// TIA Portal V17 export
// export: Created 2023-09-11T12:03:28.587249Z, ExportSetting WithDefaults, DisplayName Totally Integrated Automation Portal, DisplayVersion V17 Update 6, DisplayName TIA Portal Openness, DisplayVersion V17 Update 6, DisplayName TIA Portal Teamcenter Gateway, DisplayVersion V17 Update 6, DisplayName TIA Portal Version Control Interface, DisplayVersion V17, DisplayName Simotion SCOUT TIA, DisplayVersion 5.4.3.0, DisplayName TIA Portal Test Suite Advanced, DisplayVersion V17 Update 1, DisplayName SIMOCODE ES, DisplayVersion V17 Update 5, DisplayName SINAMICS Startdrive Advanced, DisplayVersion V17 SP1, DisplayName SINAMICS Startdrive G130, G150, S120, S150, SINAMICS MV, S210, DisplayVersion V17 SP1, DisplayName SINAMICS Startdrive G110M, G120, G120C, G120D, G120P, G115D, DisplayVersion V17 SP1, DisplayName SIRIUS Safety ES, DisplayVersion V17 Update 5, DisplayName STEP 7 Professional, DisplayVersion V17 Update 6, DisplayName STEP 7 CFC, DisplayVersion V17 Update 1, DisplayName STEP 7 Safety, DisplayVersion V17 Update 6, DisplayName WinCC Advanced, DisplayVersion V17 Update 6, DisplayName SIMATIC Visualization Architect, DisplayVersion V17 Update 5
FUNCTION "03_Zone Cumulative" : Void   // FC4, F_FBD
{ S7_Optimized_Access := 'TRUE' }
VERSION : 0.1
// stored: AutoNumber true, IsIECCheckEnabled false, UDAEnableTagReadback false
BEGIN

REGION Network 1: S1 PB - ^S1 | Sorter COY Upper [=SC01]
   // 251 - 500 Inputs
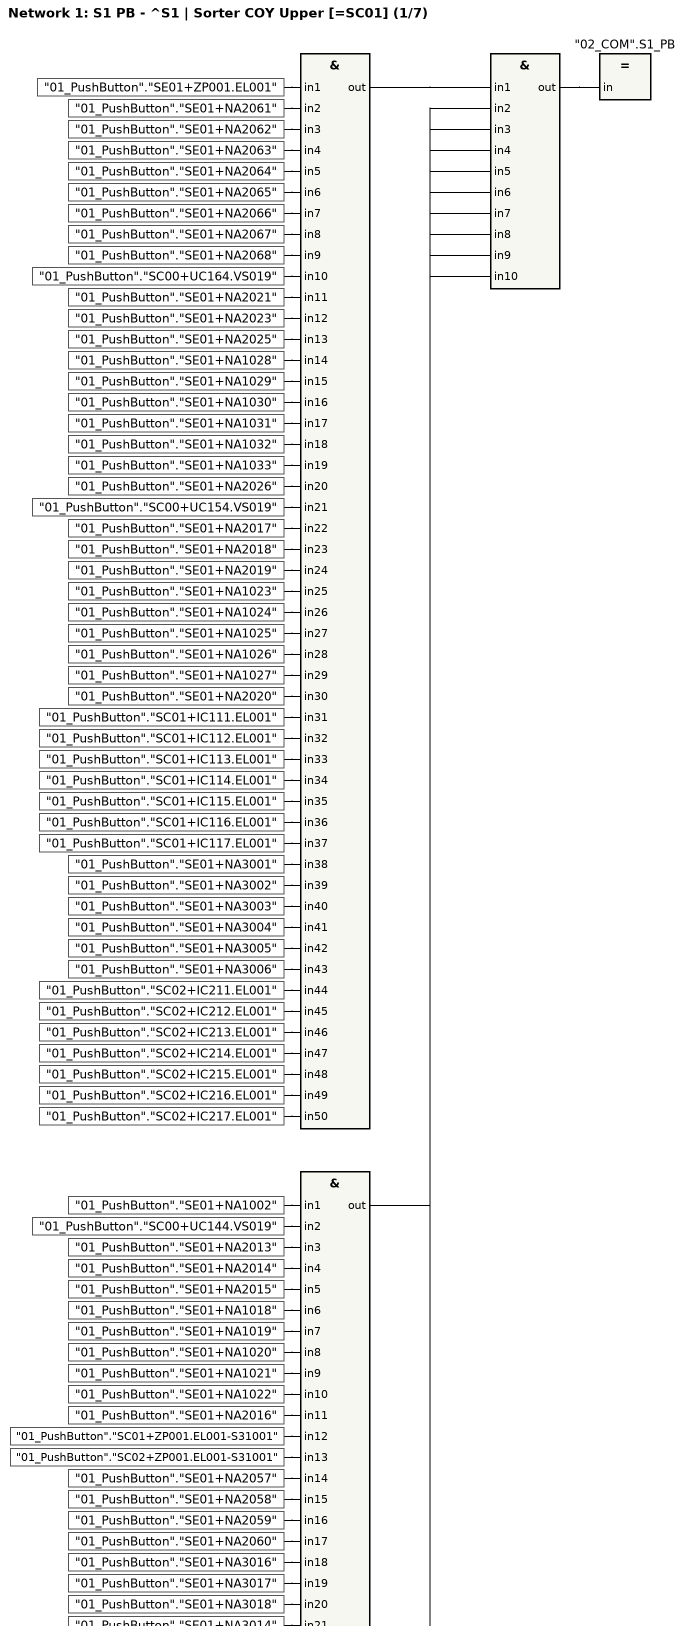
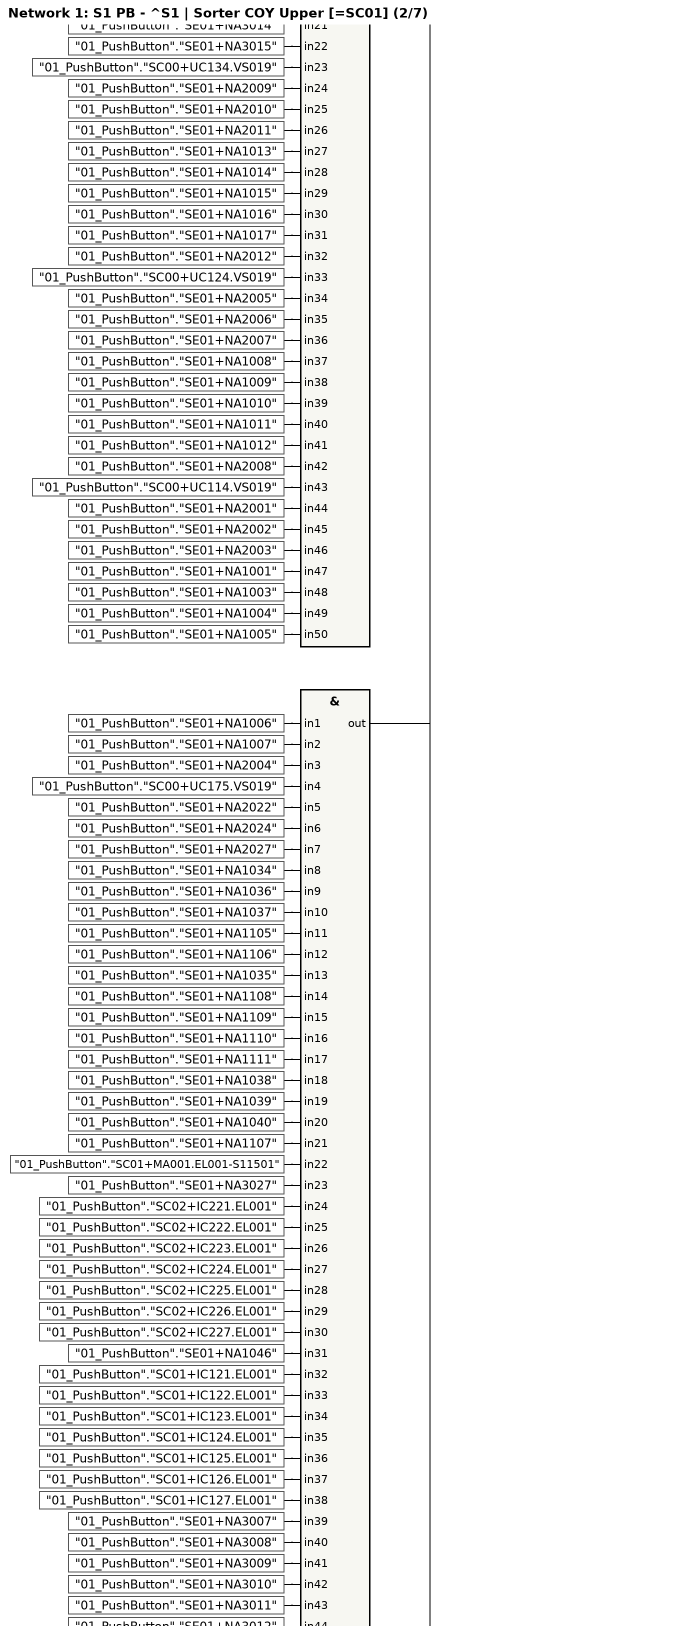
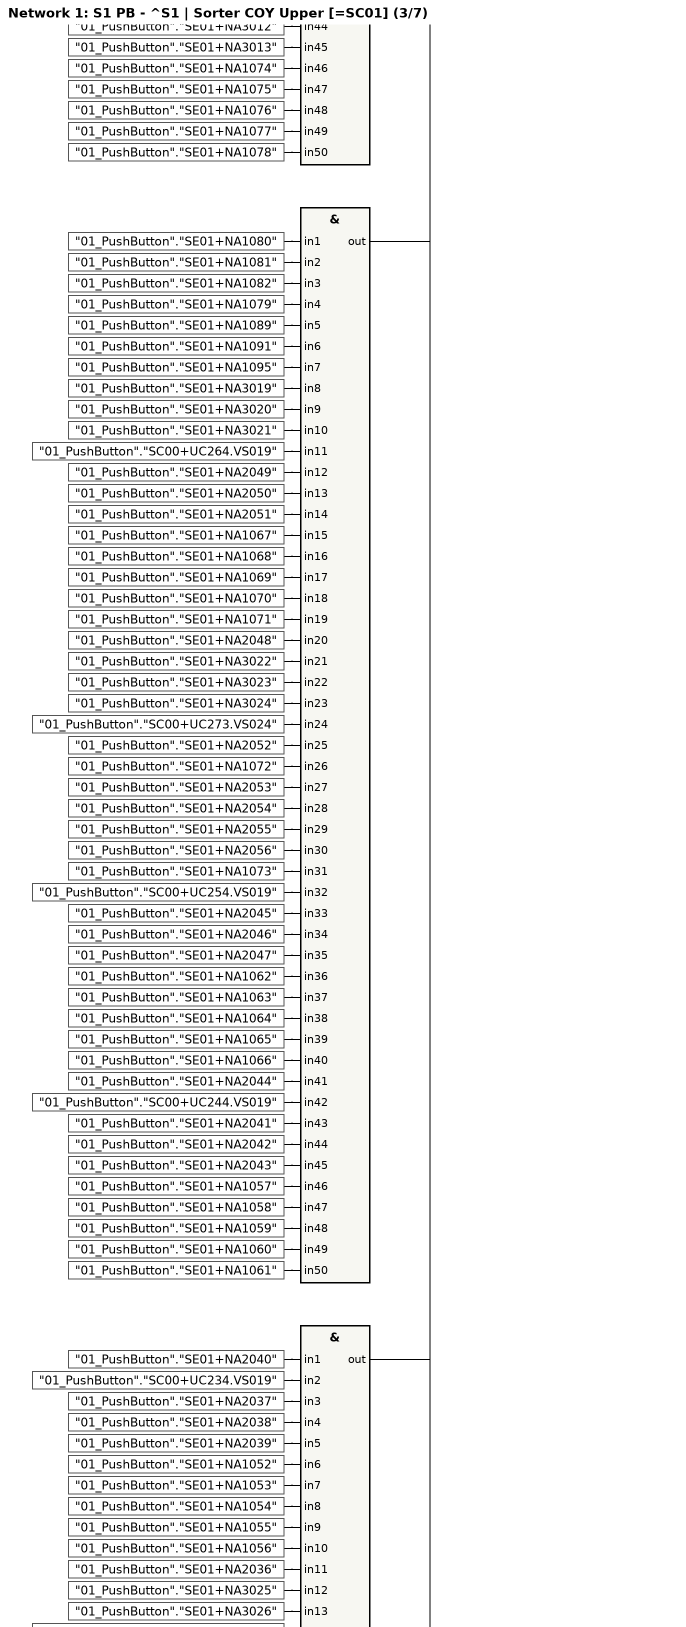
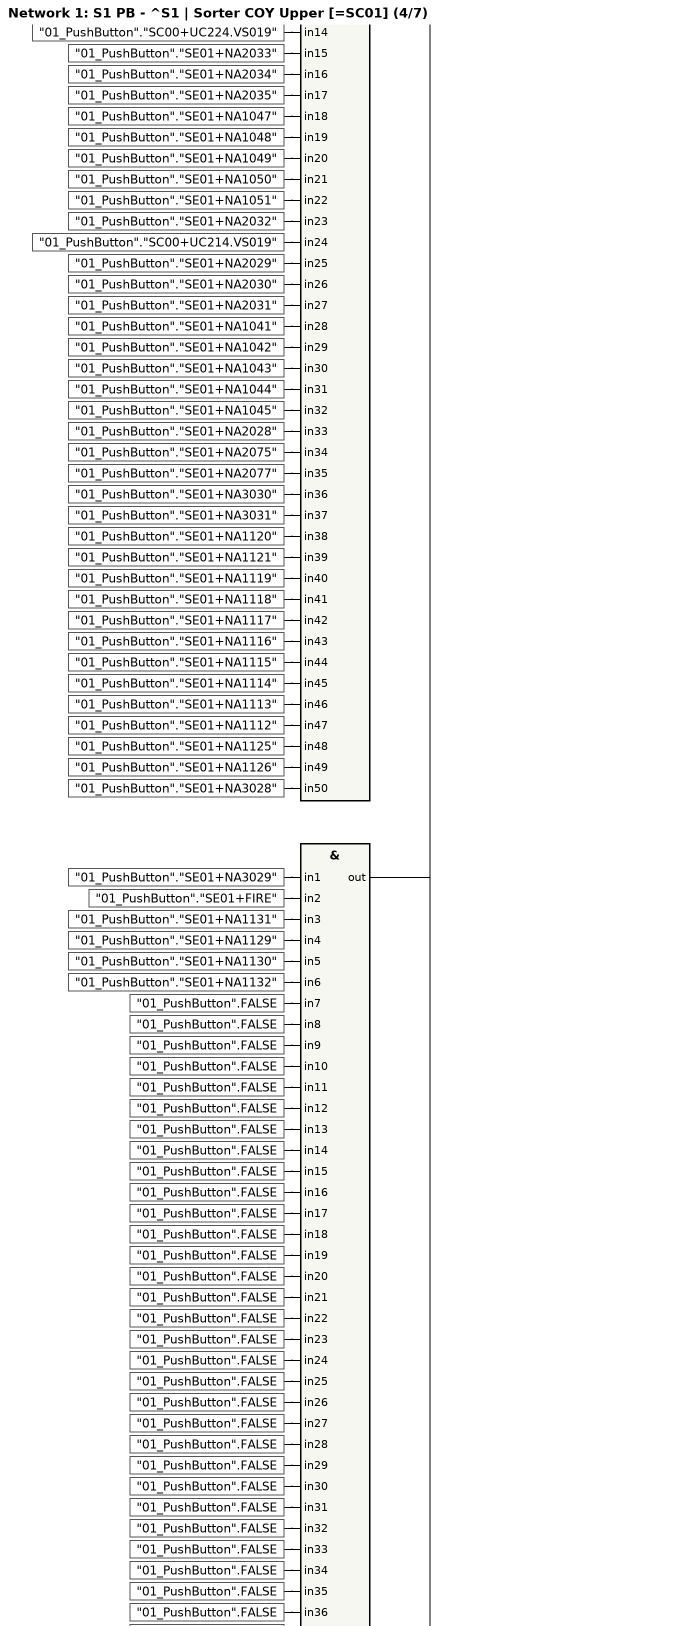
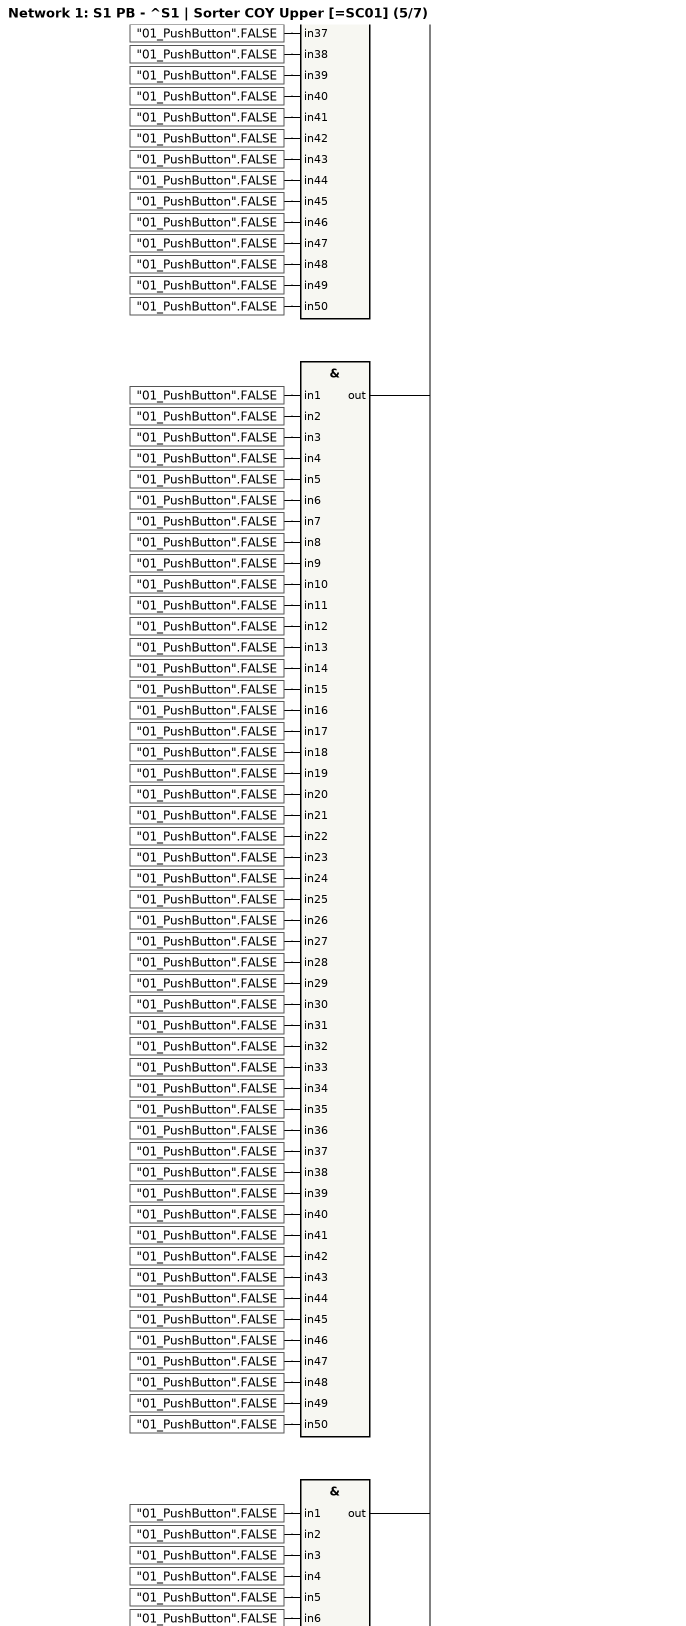
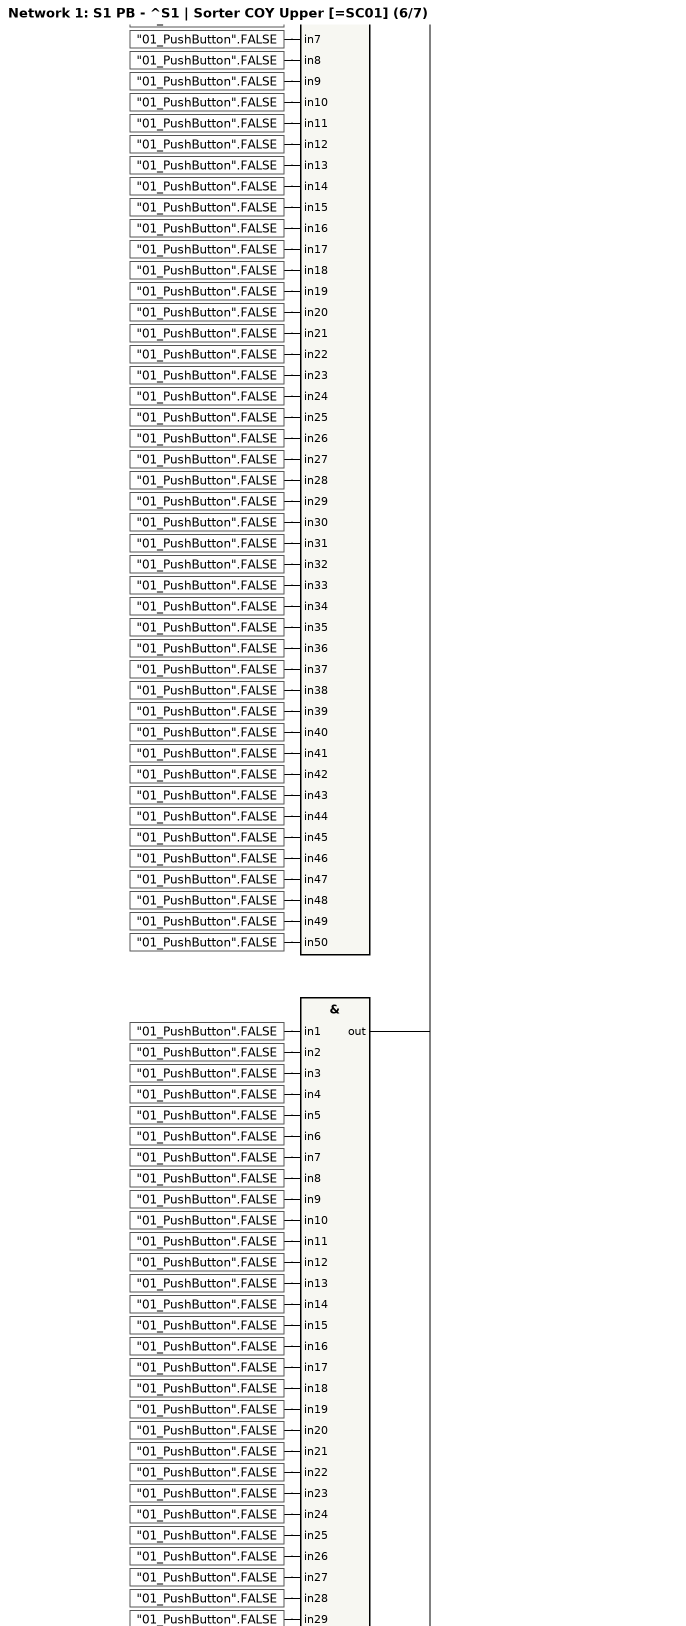
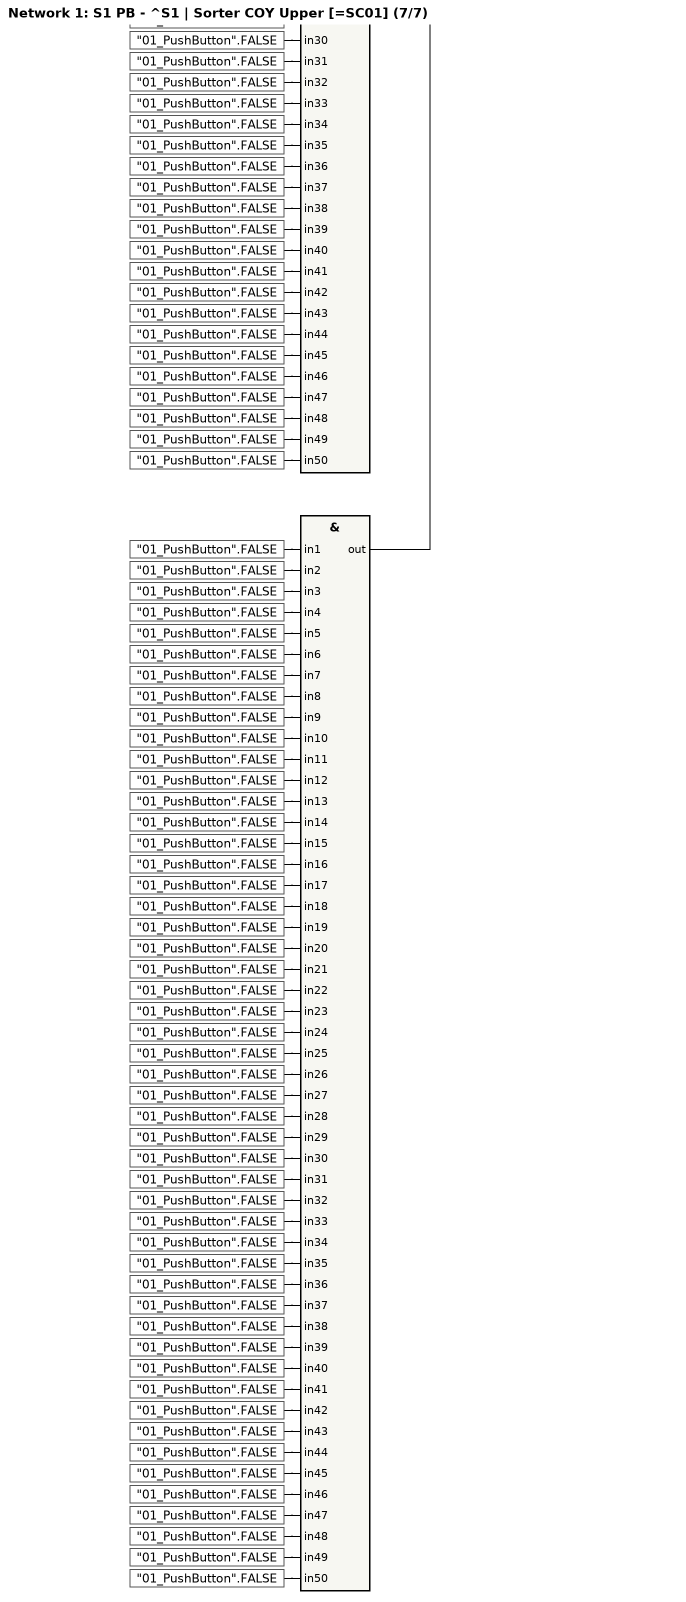
   "02_COM".S1_PB := "01_PushButton"."SE01+ZP001.EL001" AND "01_PushButton"."SE01+NA2061" AND "01_PushButton"."SE01+NA2062" AND "01_PushButton"."SE01+NA2063" AND "01_PushButton"."SE01+NA2064" AND "01_PushButton"."SE01+NA2065" AND "01_PushButton"."SE01+NA2066" AND "01_PushButton"."SE01+NA2067" AND "01_PushButton"."SE01+NA2068" AND "01_PushButton"."SC00+UC164.VS019" AND "01_PushButton"."SE01+NA2021" AND "01_PushButton"."SE01+NA2023" AND "01_PushButton"."SE01+NA2025" AND "01_PushButton"."SE01+NA1028" AND "01_PushButton"."SE01+NA1029" AND "01_PushButton"."SE01+NA1030" AND "01_PushButton"."SE01+NA1031" AND "01_PushButton"."SE01+NA1032" AND "01_PushButton"."SE01+NA1033" AND "01_PushButton"."SE01+NA2026" AND "01_PushButton"."SC00+UC154.VS019" AND "01_PushButton"."SE01+NA2017" AND "01_PushButton"."SE01+NA2018" AND "01_PushButton"."SE01+NA2019" AND "01_PushButton"."SE01+NA1023" AND "01_PushButton"."SE01+NA1024" AND "01_PushButton"."SE01+NA1025" AND "01_PushButton"."SE01+NA1026" AND "01_PushButton"."SE01+NA1027" AND "01_PushButton"."SE01+NA2020" AND "01_PushButton"."SC01+IC111.EL001" AND "01_PushButton"."SC01+IC112.EL001" AND "01_PushButton"."SC01+IC113.EL001" AND "01_PushButton"."SC01+IC114.EL001" AND "01_PushButton"."SC01+IC115.EL001" AND "01_PushButton"."SC01+IC116.EL001" AND "01_PushButton"."SC01+IC117.EL001" AND "01_PushButton"."SE01+NA3001" AND "01_PushButton"."SE01+NA3002" AND "01_PushButton"."SE01+NA3003" AND "01_PushButton"."SE01+NA3004" AND "01_PushButton"."SE01+NA3005" AND "01_PushButton"."SE01+NA3006" AND "01_PushButton"."SC02+IC211.EL001" AND "01_PushButton"."SC02+IC212.EL001" AND "01_PushButton"."SC02+IC213.EL001" AND "01_PushButton"."SC02+IC214.EL001" AND "01_PushButton"."SC02+IC215.EL001" AND "01_PushButton"."SC02+IC216.EL001" AND "01_PushButton"."SC02+IC217.EL001" AND "01_PushButton"."SE01+NA1002" AND "01_PushButton"."SC00+UC144.VS019" AND "01_PushButton"."SE01+NA2013" AND "01_PushButton"."SE01+NA2014" AND "01_PushButton"."SE01+NA2015" AND "01_PushButton"."SE01+NA1018" AND "01_PushButton"."SE01+NA1019" AND "01_PushButton"."SE01+NA1020" AND "01_PushButton"."SE01+NA1021" AND "01_PushButton"."SE01+NA1022" AND "01_PushButton"."SE01+NA2016" AND "01_PushButton"."SC01+ZP001.EL001-S31001" AND "01_PushButton"."SC02+ZP001.EL001-S31001" AND "01_PushButton"."SE01+NA2057" AND "01_PushButton"."SE01+NA2058" AND "01_PushButton"."SE01+NA2059" AND "01_PushButton"."SE01+NA2060" AND "01_PushButton"."SE01+NA3016" AND "01_PushButton"."SE01+NA3017" AND "01_PushButton"."SE01+NA3018" AND "01_PushButton"."SE01+NA3014" AND "01_PushButton"."SE01+NA3015" AND "01_PushButton"."SC00+UC134.VS019" AND "01_PushButton"."SE01+NA2009" AND "01_PushButton"."SE01+NA2010" AND "01_PushButton"."SE01+NA2011" AND "01_PushButton"."SE01+NA1013" AND "01_PushButton"."SE01+NA1014" AND "01_PushButton"."SE01+NA1015" AND "01_PushButton"."SE01+NA1016" AND "01_PushButton"."SE01+NA1017" AND "01_PushButton"."SE01+NA2012" AND "01_PushButton"."SC00+UC124.VS019" AND "01_PushButton"."SE01+NA2005" AND "01_PushButton"."SE01+NA2006" AND "01_PushButton"."SE01+NA2007" AND "01_PushButton"."SE01+NA1008" AND "01_PushButton"."SE01+NA1009" AND "01_PushButton"."SE01+NA1010" AND "01_PushButton"."SE01+NA1011" AND "01_PushButton"."SE01+NA1012" AND "01_PushButton"."SE01+NA2008" AND "01_PushButton"."SC00+UC114.VS019" AND "01_PushButton"."SE01+NA2001" AND "01_PushButton"."SE01+NA2002" AND "01_PushButton"."SE01+NA2003" AND "01_PushButton"."SE01+NA1001" AND "01_PushButton"."SE01+NA1003" AND "01_PushButton"."SE01+NA1004" AND "01_PushButton"."SE01+NA1005" AND "01_PushButton"."SE01+NA1006" AND "01_PushButton"."SE01+NA1007" AND "01_PushButton"."SE01+NA2004" AND "01_PushButton"."SC00+UC175.VS019" AND "01_PushButton"."SE01+NA2022" AND "01_PushButton"."SE01+NA2024" AND "01_PushButton"."SE01+NA2027" AND "01_PushButton"."SE01+NA1034" AND "01_PushButton"."SE01+NA1036" AND "01_PushButton"."SE01+NA1037" AND "01_PushButton"."SE01+NA1105" AND "01_PushButton"."SE01+NA1106" AND "01_PushButton"."SE01+NA1035" AND "01_PushButton"."SE01+NA1108" AND "01_PushButton"."SE01+NA1109" AND "01_PushButton"."SE01+NA1110" AND "01_PushButton"."SE01+NA1111" AND "01_PushButton"."SE01+NA1038" AND "01_PushButton"."SE01+NA1039" AND "01_PushButton"."SE01+NA1040" AND "01_PushButton"."SE01+NA1107" AND "01_PushButton"."SC01+MA001.EL001-S11501" AND "01_PushButton"."SE01+NA3027" AND "01_PushButton"."SC02+IC221.EL001" AND "01_PushButton"."SC02+IC222.EL001" AND "01_PushButton"."SC02+IC223.EL001" AND "01_PushButton"."SC02+IC224.EL001" AND "01_PushButton"."SC02+IC225.EL001" AND "01_PushButton"."SC02+IC226.EL001" AND "01_PushButton"."SC02+IC227.EL001" AND "01_PushButton"."SE01+NA1046" AND "01_PushButton"."SC01+IC121.EL001" AND "01_PushButton"."SC01+IC122.EL001" AND "01_PushButton"."SC01+IC123.EL001" AND "01_PushButton"."SC01+IC124.EL001" AND "01_PushButton"."SC01+IC125.EL001" AND "01_PushButton"."SC01+IC126.EL001" AND "01_PushButton"."SC01+IC127.EL001" AND "01_PushButton"."SE01+NA3007" AND "01_PushButton"."SE01+NA3008" AND "01_PushButton"."SE01+NA3009" AND "01_PushButton"."SE01+NA3010" AND "01_PushButton"."SE01+NA3011" AND "01_PushButton"."SE01+NA3012" AND "01_PushButton"."SE01+NA3013" AND "01_PushButton"."SE01+NA1074" AND "01_PushButton"."SE01+NA1075" AND "01_PushButton"."SE01+NA1076" AND "01_PushButton"."SE01+NA1077" AND "01_PushButton"."SE01+NA1078" AND "01_PushButton"."SE01+NA1080" AND "01_PushButton"."SE01+NA1081" AND "01_PushButton"."SE01+NA1082" AND "01_PushButton"."SE01+NA1079" AND "01_PushButton"."SE01+NA1089" AND "01_PushButton"."SE01+NA1091" AND "01_PushButton"."SE01+NA1095" AND "01_PushButton"."SE01+NA3019" AND "01_PushButton"."SE01+NA3020" AND "01_PushButton"."SE01+NA3021" AND "01_PushButton"."SC00+UC264.VS019" AND "01_PushButton"."SE01+NA2049" AND "01_PushButton"."SE01+NA2050" AND "01_PushButton"."SE01+NA2051" AND "01_PushButton"."SE01+NA1067" AND "01_PushButton"."SE01+NA1068" AND "01_PushButton"."SE01+NA1069" AND "01_PushButton"."SE01+NA1070" AND "01_PushButton"."SE01+NA1071" AND "01_PushButton"."SE01+NA2048" AND "01_PushButton"."SE01+NA3022" AND "01_PushButton"."SE01+NA3023" AND "01_PushButton"."SE01+NA3024" AND "01_PushButton"."SC00+UC273.VS024" AND "01_PushButton"."SE01+NA2052" AND "01_PushButton"."SE01+NA1072" AND "01_PushButton"."SE01+NA2053" AND "01_PushButton"."SE01+NA2054" AND "01_PushButton"."SE01+NA2055" AND "01_PushButton"."SE01+NA2056" AND "01_PushButton"."SE01+NA1073" AND "01_PushButton"."SC00+UC254.VS019" AND "01_PushButton"."SE01+NA2045" AND "01_PushButton"."SE01+NA2046" AND "01_PushButton"."SE01+NA2047" AND "01_PushButton"."SE01+NA1062" AND "01_PushButton"."SE01+NA1063" AND "01_PushButton"."SE01+NA1064" AND "01_PushButton"."SE01+NA1065" AND "01_PushButton"."SE01+NA1066" AND "01_PushButton"."SE01+NA2044" AND "01_PushButton"."SC00+UC244.VS019" AND "01_PushButton"."SE01+NA2041" AND "01_PushButton"."SE01+NA2042" AND "01_PushButton"."SE01+NA2043" AND "01_PushButton"."SE01+NA1057" AND "01_PushButton"."SE01+NA1058" AND "01_PushButton"."SE01+NA1059" AND "01_PushButton"."SE01+NA1060" AND "01_PushButton"."SE01+NA1061" AND "01_PushButton"."SE01+NA2040" AND "01_PushButton"."SC00+UC234.VS019" AND "01_PushButton"."SE01+NA2037" AND "01_PushButton"."SE01+NA2038" AND "01_PushButton"."SE01+NA2039" AND "01_PushButton"."SE01+NA1052" AND "01_PushButton"."SE01+NA1053" AND "01_PushButton"."SE01+NA1054" AND "01_PushButton"."SE01+NA1055" AND "01_PushButton"."SE01+NA1056" AND "01_PushButton"."SE01+NA2036" AND "01_PushButton"."SE01+NA3025" AND "01_PushButton"."SE01+NA3026" AND "01_PushButton"."SC00+UC224.VS019" AND "01_PushButton"."SE01+NA2033" AND "01_PushButton"."SE01+NA2034" AND "01_PushButton"."SE01+NA2035" AND "01_PushButton"."SE01+NA1047" AND "01_PushButton"."SE01+NA1048" AND "01_PushButton"."SE01+NA1049" AND "01_PushButton"."SE01+NA1050" AND "01_PushButton"."SE01+NA1051" AND "01_PushButton"."SE01+NA2032" AND "01_PushButton"."SC00+UC214.VS019" AND "01_PushButton"."SE01+NA2029" AND "01_PushButton"."SE01+NA2030" AND "01_PushButton"."SE01+NA2031" AND "01_PushButton"."SE01+NA1041" AND "01_PushButton"."SE01+NA1042" AND "01_PushButton"."SE01+NA1043" AND "01_PushButton"."SE01+NA1044" AND "01_PushButton"."SE01+NA1045" AND "01_PushButton"."SE01+NA2028" AND "01_PushButton"."SE01+NA2075" AND "01_PushButton"."SE01+NA2077" AND "01_PushButton"."SE01+NA3030" AND "01_PushButton"."SE01+NA3031" AND "01_PushButton"."SE01+NA1120" AND "01_PushButton"."SE01+NA1121" AND "01_PushButton"."SE01+NA1119" AND "01_PushButton"."SE01+NA1118" AND "01_PushButton"."SE01+NA1117" AND "01_PushButton"."SE01+NA1116" AND "01_PushButton"."SE01+NA1115" AND "01_PushButton"."SE01+NA1114" AND "01_PushButton"."SE01+NA1113" AND "01_PushButton"."SE01+NA1112" AND "01_PushButton"."SE01+NA1125" AND "01_PushButton"."SE01+NA1126" AND "01_PushButton"."SE01+NA3028" AND "01_PushButton"."SE01+NA3029" AND "01_PushButton"."SE01+FIRE" AND "01_PushButton"."SE01+NA1131" AND "01_PushButton"."SE01+NA1129" AND "01_PushButton"."SE01+NA1130" AND "01_PushButton"."SE01+NA1132" AND "01_PushButton".FALSE AND "01_PushButton".FALSE AND "01_PushButton".FALSE AND "01_PushButton".FALSE AND "01_PushButton".FALSE AND "01_PushButton".FALSE AND "01_PushButton".FALSE AND "01_PushButton".FALSE AND "01_PushButton".FALSE AND "01_PushButton".FALSE AND "01_PushButton".FALSE AND "01_PushButton".FALSE AND "01_PushButton".FALSE AND "01_PushButton".FALSE AND "01_PushButton".FALSE AND "01_PushButton".FALSE AND "01_PushButton".FALSE AND "01_PushButton".FALSE AND "01_PushButton".FALSE AND "01_PushButton".FALSE AND "01_PushButton".FALSE AND "01_PushButton".FALSE AND "01_PushButton".FALSE AND "01_PushButton".FALSE AND "01_PushButton".FALSE AND "01_PushButton".FALSE AND "01_PushButton".FALSE AND "01_PushButton".FALSE AND "01_PushButton".FALSE AND "01_PushButton".FALSE AND "01_PushButton".FALSE AND "01_PushButton".FALSE AND "01_PushButton".FALSE AND "01_PushButton".FALSE AND "01_PushButton".FALSE AND "01_PushButton".FALSE AND "01_PushButton".FALSE AND "01_PushButton".FALSE AND "01_PushButton".FALSE AND "01_PushButton".FALSE AND "01_PushButton".FALSE AND "01_PushButton".FALSE AND "01_PushButton".FALSE AND "01_PushButton".FALSE AND "01_PushButton".FALSE AND "01_PushButton".FALSE AND "01_PushButton".FALSE AND "01_PushButton".FALSE AND "01_PushButton".FALSE AND "01_PushButton".FALSE AND "01_PushButton".FALSE AND "01_PushButton".FALSE AND "01_PushButton".FALSE AND "01_PushButton".FALSE AND "01_PushButton".FALSE AND "01_PushButton".FALSE AND "01_PushButton".FALSE AND "01_PushButton".FALSE AND "01_PushButton".FALSE AND "01_PushButton".FALSE AND "01_PushButton".FALSE AND "01_PushButton".FALSE AND "01_PushButton".FALSE AND "01_PushButton".FALSE AND "01_PushButton".FALSE AND "01_PushButton".FALSE AND "01_PushButton".FALSE AND "01_PushButton".FALSE AND "01_PushButton".FALSE AND "01_PushButton".FALSE AND "01_PushButton".FALSE AND "01_PushButton".FALSE AND "01_PushButton".FALSE AND "01_PushButton".FALSE AND "01_PushButton".FALSE AND "01_PushButton".FALSE AND "01_PushButton".FALSE AND "01_PushButton".FALSE AND "01_PushButton".FALSE AND "01_PushButton".FALSE AND "01_PushButton".FALSE AND "01_PushButton".FALSE AND "01_PushButton".FALSE AND "01_PushButton".FALSE AND "01_PushButton".FALSE AND "01_PushButton".FALSE AND "01_PushButton".FALSE AND "01_PushButton".FALSE AND "01_PushButton".FALSE AND "01_PushButton".FALSE AND "01_PushButton".FALSE AND "01_PushButton".FALSE AND "01_PushButton".FALSE AND "01_PushButton".FALSE AND "01_PushButton".FALSE AND "01_PushButton".FALSE AND "01_PushButton".FALSE AND "01_PushButton".FALSE AND "01_PushButton".FALSE AND "01_PushButton".FALSE AND "01_PushButton".FALSE AND "01_PushButton".FALSE AND "01_PushButton".FALSE AND "01_PushButton".FALSE AND "01_PushButton".FALSE AND "01_PushButton".FALSE AND "01_PushButton".FALSE AND "01_PushButton".FALSE AND "01_PushButton".FALSE AND "01_PushButton".FALSE AND "01_PushButton".FALSE AND "01_PushButton".FALSE AND "01_PushButton".FALSE AND "01_PushButton".FALSE AND "01_PushButton".FALSE AND "01_PushButton".FALSE AND "01_PushButton".FALSE AND "01_PushButton".FALSE AND "01_PushButton".FALSE AND "01_PushButton".FALSE AND "01_PushButton".FALSE AND "01_PushButton".FALSE AND "01_PushButton".FALSE AND "01_PushButton".FALSE AND "01_PushButton".FALSE AND "01_PushButton".FALSE AND "01_PushButton".FALSE AND "01_PushButton".FALSE AND "01_PushButton".FALSE AND "01_PushButton".FALSE AND "01_PushButton".FALSE AND "01_PushButton".FALSE AND "01_PushButton".FALSE AND "01_PushButton".FALSE AND "01_PushButton".FALSE AND "01_PushButton".FALSE AND "01_PushButton".FALSE AND "01_PushButton".FALSE AND "01_PushButton".FALSE AND "01_PushButton".FALSE AND "01_PushButton".FALSE AND "01_PushButton".FALSE AND "01_PushButton".FALSE AND "01_PushButton".FALSE AND "01_PushButton".FALSE AND "01_PushButton".FALSE AND "01_PushButton".FALSE AND "01_PushButton".FALSE AND "01_PushButton".FALSE AND "01_PushButton".FALSE AND "01_PushButton".FALSE AND "01_PushButton".FALSE AND "01_PushButton".FALSE AND "01_PushButton".FALSE AND "01_PushButton".FALSE AND "01_PushButton".FALSE AND "01_PushButton".FALSE AND "01_PushButton".FALSE AND "01_PushButton".FALSE AND "01_PushButton".FALSE AND "01_PushButton".FALSE AND "01_PushButton".FALSE AND "01_PushButton".FALSE AND "01_PushButton".FALSE AND "01_PushButton".FALSE AND "01_PushButton".FALSE AND "01_PushButton".FALSE AND "01_PushButton".FALSE AND "01_PushButton".FALSE AND "01_PushButton".FALSE AND "01_PushButton".FALSE AND "01_PushButton".FALSE AND "01_PushButton".FALSE AND "01_PushButton".FALSE AND "01_PushButton".FALSE AND "01_PushButton".FALSE AND "01_PushButton".FALSE AND "01_PushButton".FALSE AND "01_PushButton".FALSE AND "01_PushButton".FALSE AND "01_PushButton".FALSE AND "01_PushButton".FALSE AND "01_PushButton".FALSE AND "01_PushButton".FALSE AND "01_PushButton".FALSE AND "01_PushButton".FALSE AND "01_PushButton".FALSE AND "01_PushButton".FALSE AND "01_PushButton".FALSE AND "01_PushButton".FALSE AND "01_PushButton".FALSE AND "01_PushButton".FALSE AND "01_PushButton".FALSE AND "01_PushButton".FALSE AND "01_PushButton".FALSE AND "01_PushButton".FALSE AND "01_PushButton".FALSE AND "01_PushButton".FALSE AND "01_PushButton".FALSE AND "01_PushButton".FALSE AND "01_PushButton".FALSE AND "01_PushButton".FALSE AND "01_PushButton".FALSE AND "01_PushButton".FALSE AND "01_PushButton".FALSE AND "01_PushButton".FALSE AND "01_PushButton".FALSE AND "01_PushButton".FALSE AND "01_PushButton".FALSE AND "01_PushButton".FALSE AND "01_PushButton".FALSE AND "01_PushButton".FALSE AND "01_PushButton".FALSE AND "01_PushButton".FALSE AND "01_PushButton".FALSE AND "01_PushButton".FALSE AND "01_PushButton".FALSE AND "01_PushButton".FALSE AND "01_PushButton".FALSE AND "01_PushButton".FALSE AND "01_PushButton".FALSE AND "01_PushButton".FALSE AND "01_PushButton".FALSE AND "01_PushButton".FALSE AND "01_PushButton".FALSE AND "01_PushButton".FALSE AND "01_PushButton".FALSE AND "01_PushButton".FALSE AND "01_PushButton".FALSE AND "01_PushButton".FALSE AND "01_PushButton".FALSE AND "01_PushButton".FALSE AND "01_PushButton".FALSE AND "01_PushButton".FALSE AND "01_PushButton".FALSE AND "01_PushButton".FALSE AND "01_PushButton".FALSE AND "01_PushButton".FALSE AND "01_PushButton".FALSE AND "01_PushButton".FALSE AND "01_PushButton".FALSE AND "01_PushButton".FALSE AND "01_PushButton".FALSE AND "01_PushButton".FALSE;
END_REGION

REGION Network 2: S2 PB - ^S2 | Sorter COY Lower [=SC02]
   // 251 - 500 Inputs
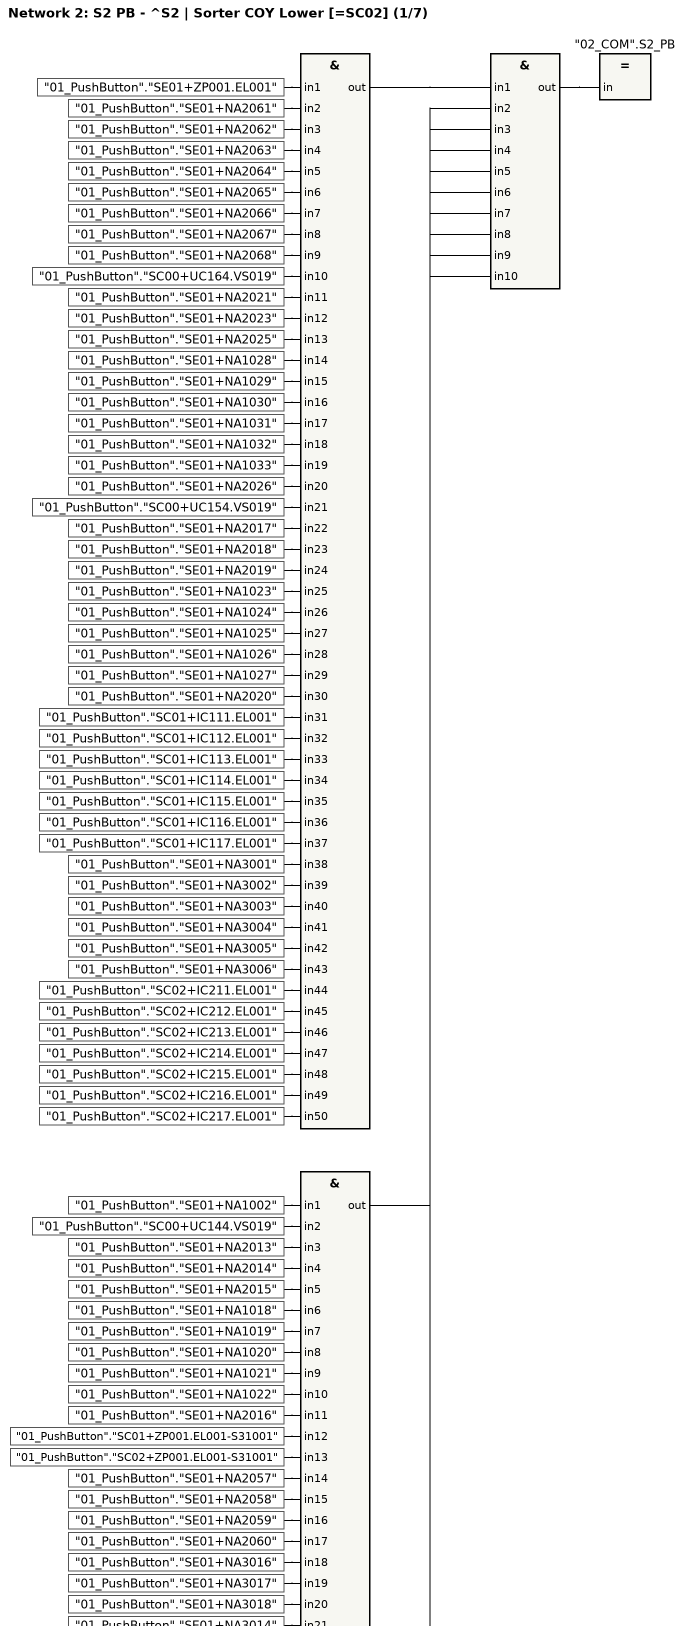
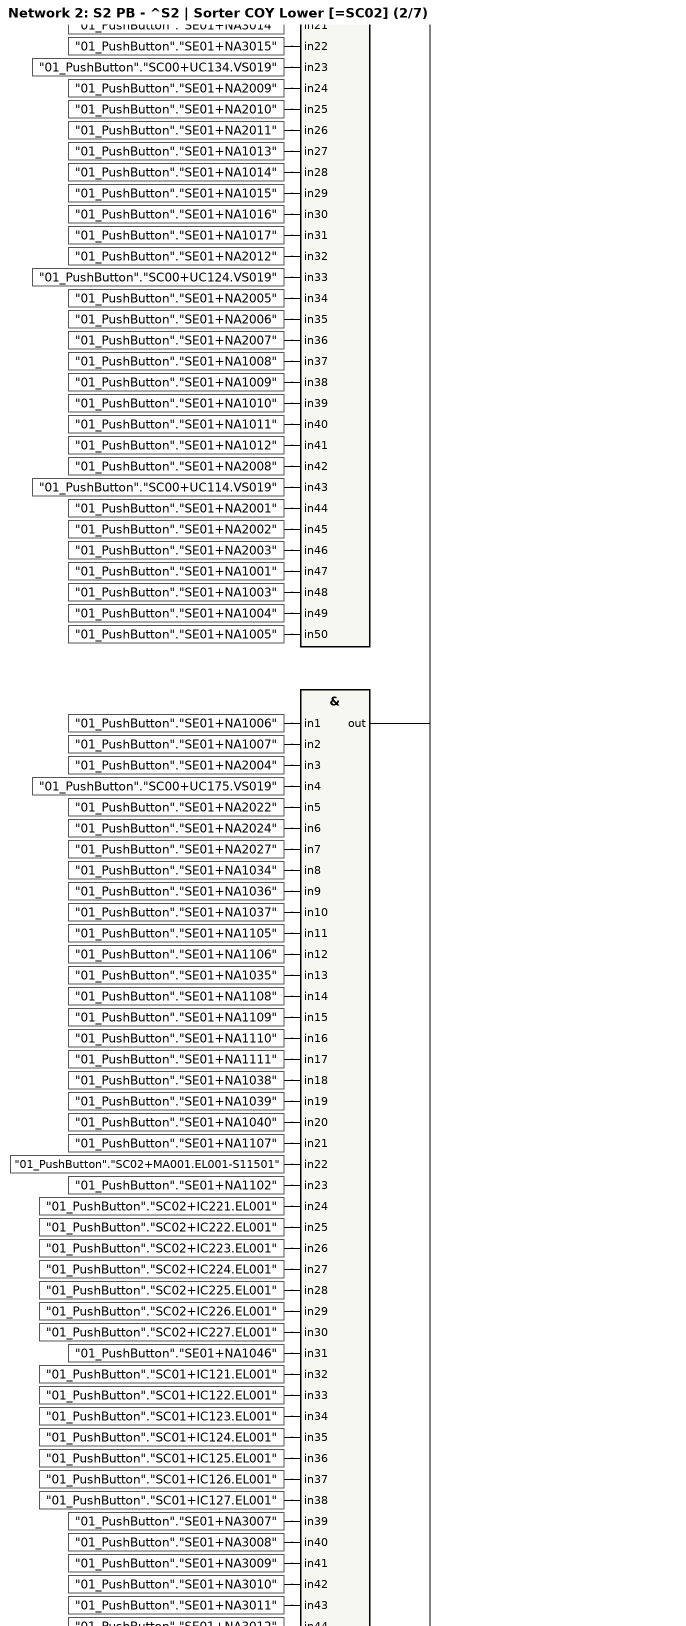
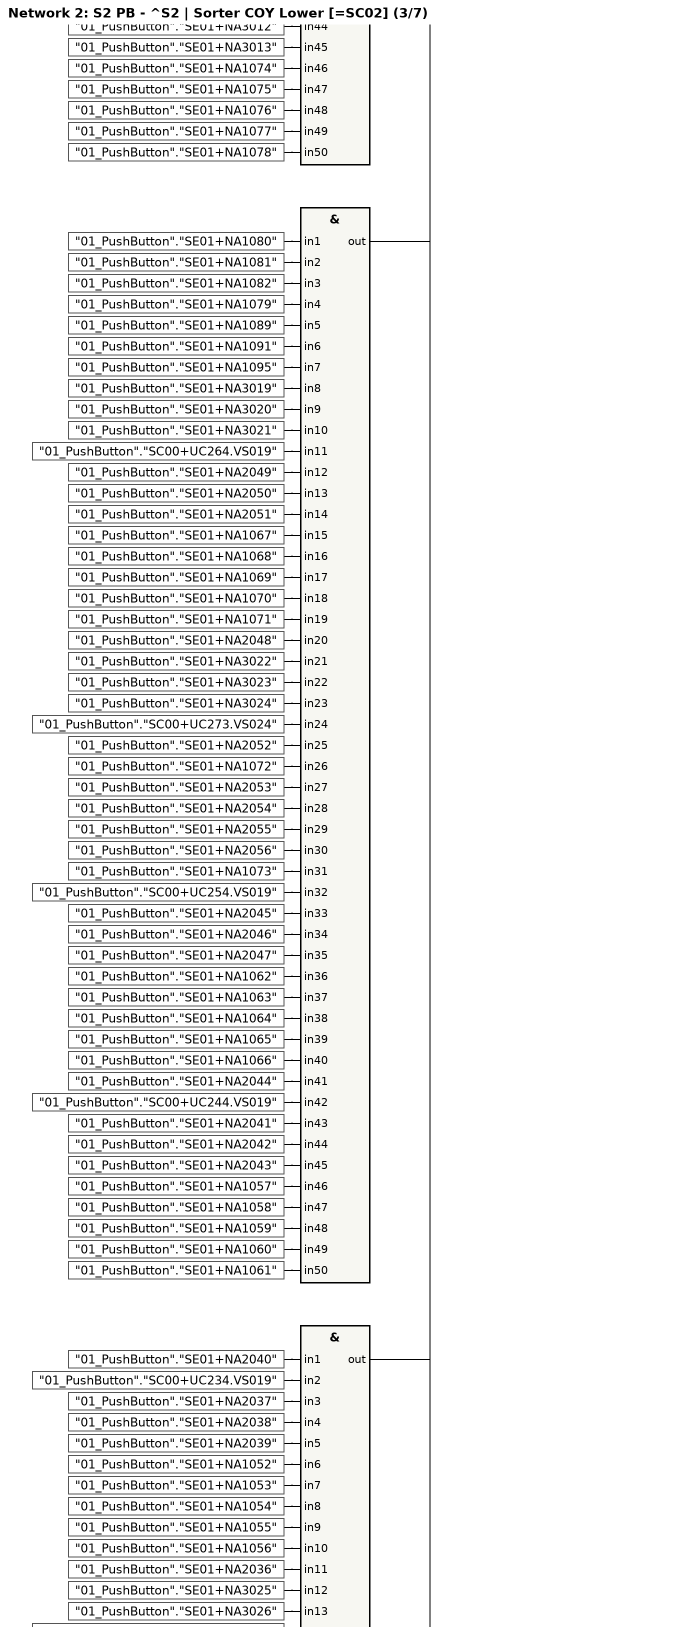
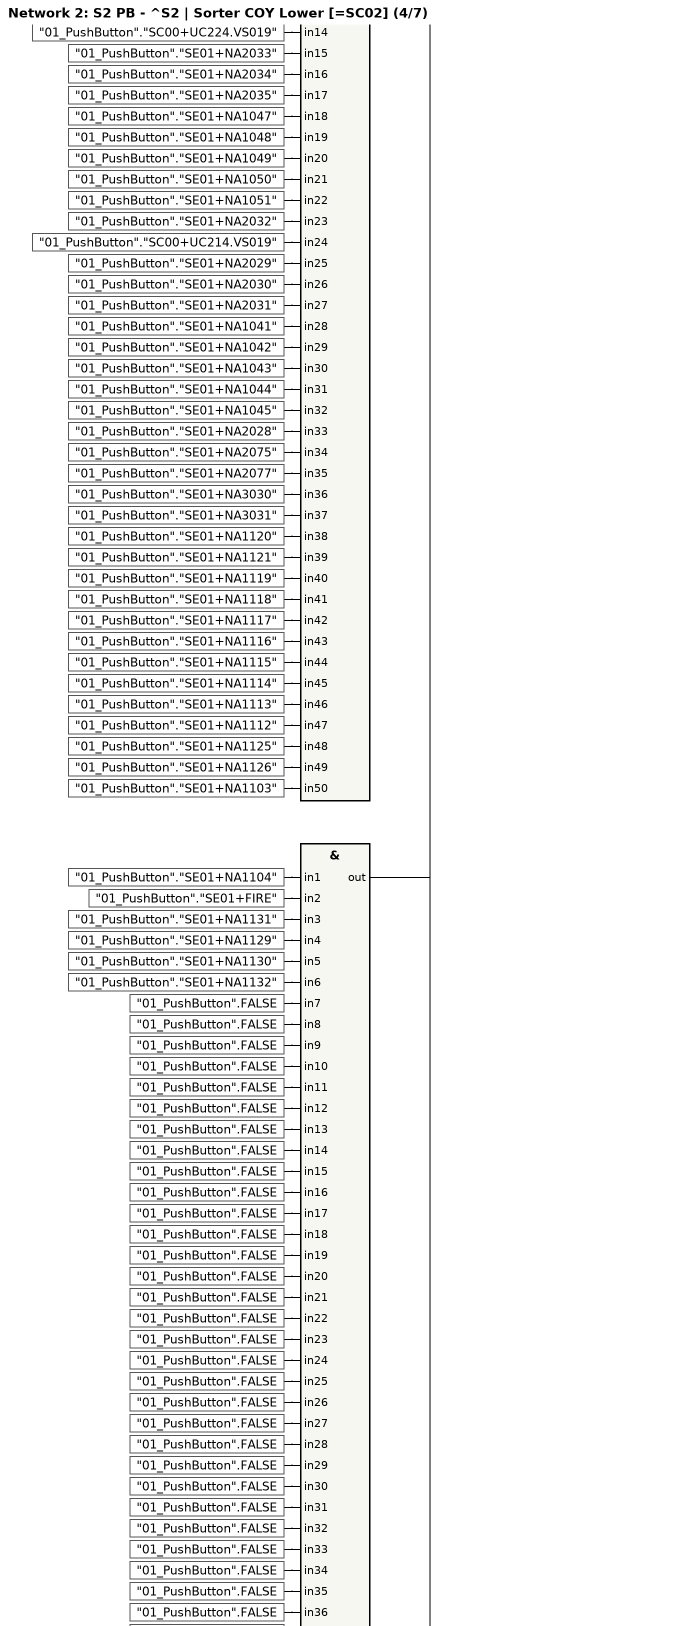
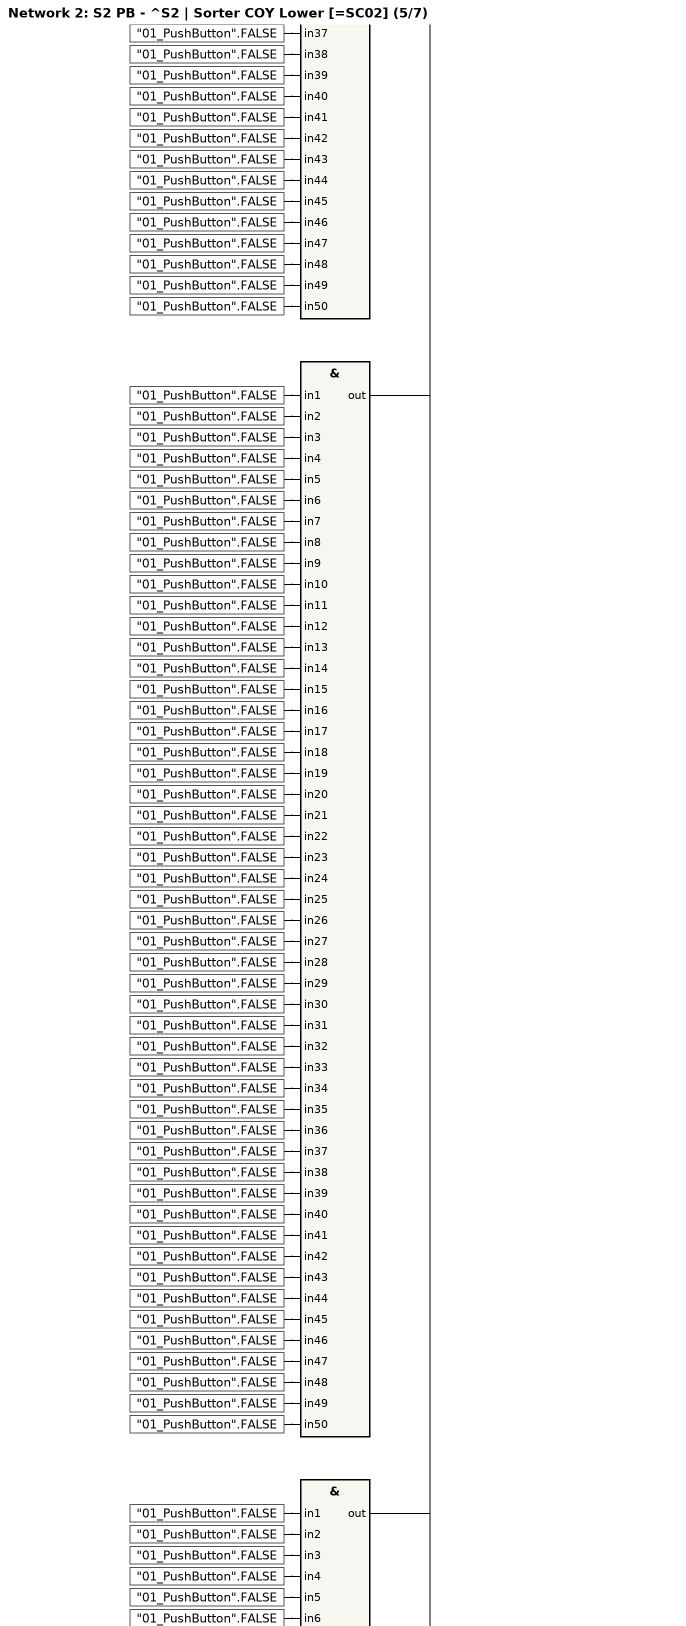
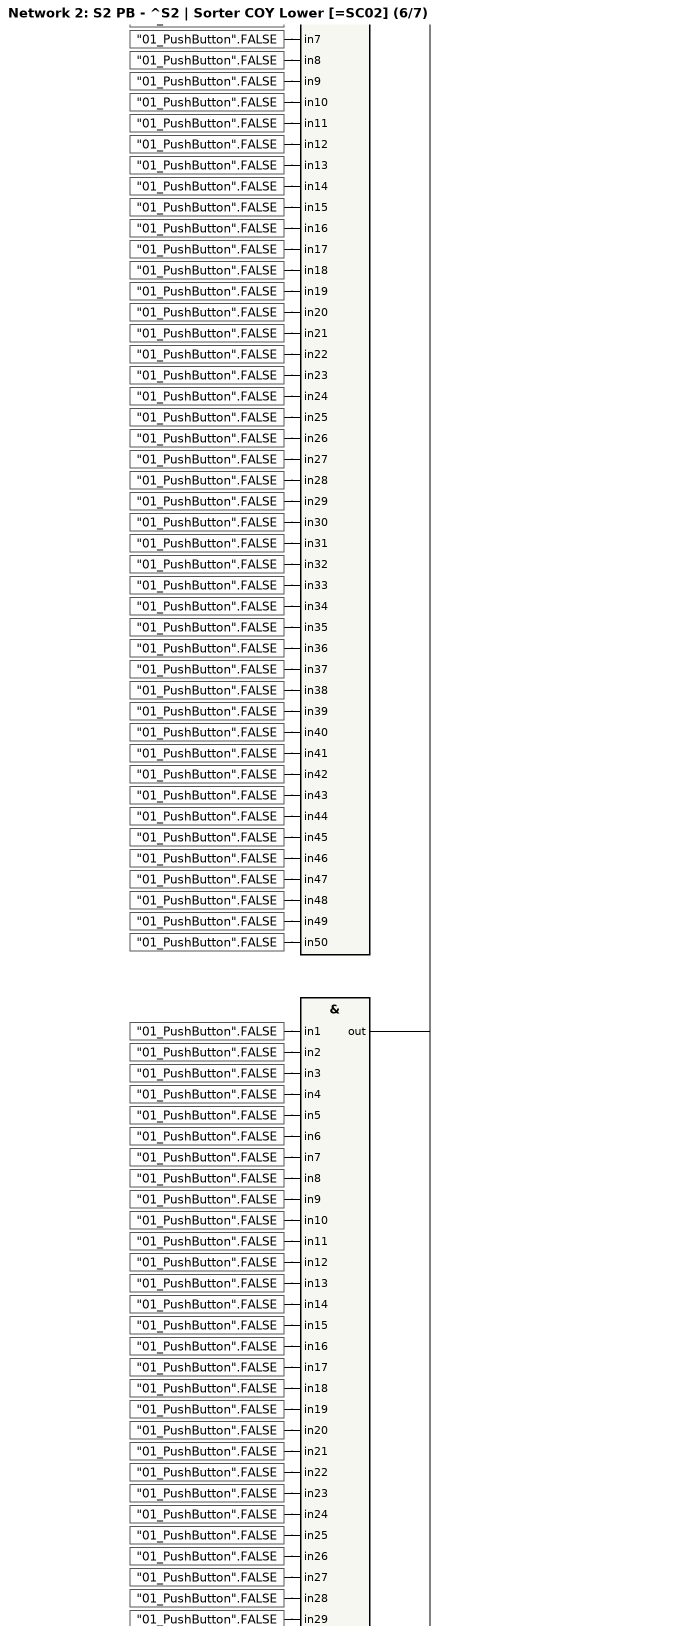
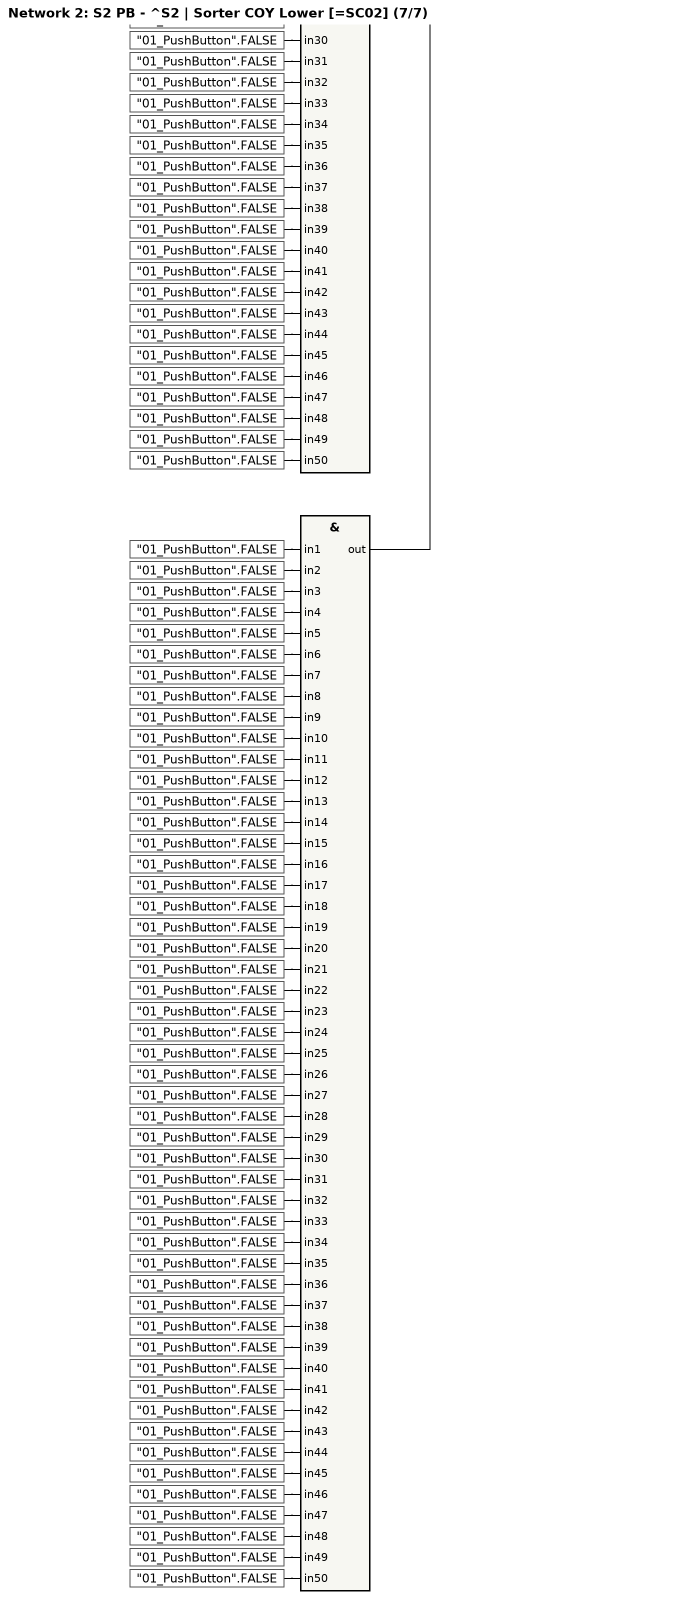
   "02_COM".S2_PB := "01_PushButton"."SE01+ZP001.EL001" AND "01_PushButton"."SE01+NA2061" AND "01_PushButton"."SE01+NA2062" AND "01_PushButton"."SE01+NA2063" AND "01_PushButton"."SE01+NA2064" AND "01_PushButton"."SE01+NA2065" AND "01_PushButton"."SE01+NA2066" AND "01_PushButton"."SE01+NA2067" AND "01_PushButton"."SE01+NA2068" AND "01_PushButton"."SC00+UC164.VS019" AND "01_PushButton"."SE01+NA2021" AND "01_PushButton"."SE01+NA2023" AND "01_PushButton"."SE01+NA2025" AND "01_PushButton"."SE01+NA1028" AND "01_PushButton"."SE01+NA1029" AND "01_PushButton"."SE01+NA1030" AND "01_PushButton"."SE01+NA1031" AND "01_PushButton"."SE01+NA1032" AND "01_PushButton"."SE01+NA1033" AND "01_PushButton"."SE01+NA2026" AND "01_PushButton"."SC00+UC154.VS019" AND "01_PushButton"."SE01+NA2017" AND "01_PushButton"."SE01+NA2018" AND "01_PushButton"."SE01+NA2019" AND "01_PushButton"."SE01+NA1023" AND "01_PushButton"."SE01+NA1024" AND "01_PushButton"."SE01+NA1025" AND "01_PushButton"."SE01+NA1026" AND "01_PushButton"."SE01+NA1027" AND "01_PushButton"."SE01+NA2020" AND "01_PushButton"."SC01+IC111.EL001" AND "01_PushButton"."SC01+IC112.EL001" AND "01_PushButton"."SC01+IC113.EL001" AND "01_PushButton"."SC01+IC114.EL001" AND "01_PushButton"."SC01+IC115.EL001" AND "01_PushButton"."SC01+IC116.EL001" AND "01_PushButton"."SC01+IC117.EL001" AND "01_PushButton"."SE01+NA3001" AND "01_PushButton"."SE01+NA3002" AND "01_PushButton"."SE01+NA3003" AND "01_PushButton"."SE01+NA3004" AND "01_PushButton"."SE01+NA3005" AND "01_PushButton"."SE01+NA3006" AND "01_PushButton"."SC02+IC211.EL001" AND "01_PushButton"."SC02+IC212.EL001" AND "01_PushButton"."SC02+IC213.EL001" AND "01_PushButton"."SC02+IC214.EL001" AND "01_PushButton"."SC02+IC215.EL001" AND "01_PushButton"."SC02+IC216.EL001" AND "01_PushButton"."SC02+IC217.EL001" AND "01_PushButton"."SE01+NA1002" AND "01_PushButton"."SC00+UC144.VS019" AND "01_PushButton"."SE01+NA2013" AND "01_PushButton"."SE01+NA2014" AND "01_PushButton"."SE01+NA2015" AND "01_PushButton"."SE01+NA1018" AND "01_PushButton"."SE01+NA1019" AND "01_PushButton"."SE01+NA1020" AND "01_PushButton"."SE01+NA1021" AND "01_PushButton"."SE01+NA1022" AND "01_PushButton"."SE01+NA2016" AND "01_PushButton"."SC01+ZP001.EL001-S31001" AND "01_PushButton"."SC02+ZP001.EL001-S31001" AND "01_PushButton"."SE01+NA2057" AND "01_PushButton"."SE01+NA2058" AND "01_PushButton"."SE01+NA2059" AND "01_PushButton"."SE01+NA2060" AND "01_PushButton"."SE01+NA3016" AND "01_PushButton"."SE01+NA3017" AND "01_PushButton"."SE01+NA3018" AND "01_PushButton"."SE01+NA3014" AND "01_PushButton"."SE01+NA3015" AND "01_PushButton"."SC00+UC134.VS019" AND "01_PushButton"."SE01+NA2009" AND "01_PushButton"."SE01+NA2010" AND "01_PushButton"."SE01+NA2011" AND "01_PushButton"."SE01+NA1013" AND "01_PushButton"."SE01+NA1014" AND "01_PushButton"."SE01+NA1015" AND "01_PushButton"."SE01+NA1016" AND "01_PushButton"."SE01+NA1017" AND "01_PushButton"."SE01+NA2012" AND "01_PushButton"."SC00+UC124.VS019" AND "01_PushButton"."SE01+NA2005" AND "01_PushButton"."SE01+NA2006" AND "01_PushButton"."SE01+NA2007" AND "01_PushButton"."SE01+NA1008" AND "01_PushButton"."SE01+NA1009" AND "01_PushButton"."SE01+NA1010" AND "01_PushButton"."SE01+NA1011" AND "01_PushButton"."SE01+NA1012" AND "01_PushButton"."SE01+NA2008" AND "01_PushButton"."SC00+UC114.VS019" AND "01_PushButton"."SE01+NA2001" AND "01_PushButton"."SE01+NA2002" AND "01_PushButton"."SE01+NA2003" AND "01_PushButton"."SE01+NA1001" AND "01_PushButton"."SE01+NA1003" AND "01_PushButton"."SE01+NA1004" AND "01_PushButton"."SE01+NA1005" AND "01_PushButton"."SE01+NA1006" AND "01_PushButton"."SE01+NA1007" AND "01_PushButton"."SE01+NA2004" AND "01_PushButton"."SC00+UC175.VS019" AND "01_PushButton"."SE01+NA2022" AND "01_PushButton"."SE01+NA2024" AND "01_PushButton"."SE01+NA2027" AND "01_PushButton"."SE01+NA1034" AND "01_PushButton"."SE01+NA1036" AND "01_PushButton"."SE01+NA1037" AND "01_PushButton"."SE01+NA1105" AND "01_PushButton"."SE01+NA1106" AND "01_PushButton"."SE01+NA1035" AND "01_PushButton"."SE01+NA1108" AND "01_PushButton"."SE01+NA1109" AND "01_PushButton"."SE01+NA1110" AND "01_PushButton"."SE01+NA1111" AND "01_PushButton"."SE01+NA1038" AND "01_PushButton"."SE01+NA1039" AND "01_PushButton"."SE01+NA1040" AND "01_PushButton"."SE01+NA1107" AND "01_PushButton"."SC02+MA001.EL001-S11501" AND "01_PushButton"."SE01+NA1102" AND "01_PushButton"."SC02+IC221.EL001" AND "01_PushButton"."SC02+IC222.EL001" AND "01_PushButton"."SC02+IC223.EL001" AND "01_PushButton"."SC02+IC224.EL001" AND "01_PushButton"."SC02+IC225.EL001" AND "01_PushButton"."SC02+IC226.EL001" AND "01_PushButton"."SC02+IC227.EL001" AND "01_PushButton"."SE01+NA1046" AND "01_PushButton"."SC01+IC121.EL001" AND "01_PushButton"."SC01+IC122.EL001" AND "01_PushButton"."SC01+IC123.EL001" AND "01_PushButton"."SC01+IC124.EL001" AND "01_PushButton"."SC01+IC125.EL001" AND "01_PushButton"."SC01+IC126.EL001" AND "01_PushButton"."SC01+IC127.EL001" AND "01_PushButton"."SE01+NA3007" AND "01_PushButton"."SE01+NA3008" AND "01_PushButton"."SE01+NA3009" AND "01_PushButton"."SE01+NA3010" AND "01_PushButton"."SE01+NA3011" AND "01_PushButton"."SE01+NA3012" AND "01_PushButton"."SE01+NA3013" AND "01_PushButton"."SE01+NA1074" AND "01_PushButton"."SE01+NA1075" AND "01_PushButton"."SE01+NA1076" AND "01_PushButton"."SE01+NA1077" AND "01_PushButton"."SE01+NA1078" AND "01_PushButton"."SE01+NA1080" AND "01_PushButton"."SE01+NA1081" AND "01_PushButton"."SE01+NA1082" AND "01_PushButton"."SE01+NA1079" AND "01_PushButton"."SE01+NA1089" AND "01_PushButton"."SE01+NA1091" AND "01_PushButton"."SE01+NA1095" AND "01_PushButton"."SE01+NA3019" AND "01_PushButton"."SE01+NA3020" AND "01_PushButton"."SE01+NA3021" AND "01_PushButton"."SC00+UC264.VS019" AND "01_PushButton"."SE01+NA2049" AND "01_PushButton"."SE01+NA2050" AND "01_PushButton"."SE01+NA2051" AND "01_PushButton"."SE01+NA1067" AND "01_PushButton"."SE01+NA1068" AND "01_PushButton"."SE01+NA1069" AND "01_PushButton"."SE01+NA1070" AND "01_PushButton"."SE01+NA1071" AND "01_PushButton"."SE01+NA2048" AND "01_PushButton"."SE01+NA3022" AND "01_PushButton"."SE01+NA3023" AND "01_PushButton"."SE01+NA3024" AND "01_PushButton"."SC00+UC273.VS024" AND "01_PushButton"."SE01+NA2052" AND "01_PushButton"."SE01+NA1072" AND "01_PushButton"."SE01+NA2053" AND "01_PushButton"."SE01+NA2054" AND "01_PushButton"."SE01+NA2055" AND "01_PushButton"."SE01+NA2056" AND "01_PushButton"."SE01+NA1073" AND "01_PushButton"."SC00+UC254.VS019" AND "01_PushButton"."SE01+NA2045" AND "01_PushButton"."SE01+NA2046" AND "01_PushButton"."SE01+NA2047" AND "01_PushButton"."SE01+NA1062" AND "01_PushButton"."SE01+NA1063" AND "01_PushButton"."SE01+NA1064" AND "01_PushButton"."SE01+NA1065" AND "01_PushButton"."SE01+NA1066" AND "01_PushButton"."SE01+NA2044" AND "01_PushButton"."SC00+UC244.VS019" AND "01_PushButton"."SE01+NA2041" AND "01_PushButton"."SE01+NA2042" AND "01_PushButton"."SE01+NA2043" AND "01_PushButton"."SE01+NA1057" AND "01_PushButton"."SE01+NA1058" AND "01_PushButton"."SE01+NA1059" AND "01_PushButton"."SE01+NA1060" AND "01_PushButton"."SE01+NA1061" AND "01_PushButton"."SE01+NA2040" AND "01_PushButton"."SC00+UC234.VS019" AND "01_PushButton"."SE01+NA2037" AND "01_PushButton"."SE01+NA2038" AND "01_PushButton"."SE01+NA2039" AND "01_PushButton"."SE01+NA1052" AND "01_PushButton"."SE01+NA1053" AND "01_PushButton"."SE01+NA1054" AND "01_PushButton"."SE01+NA1055" AND "01_PushButton"."SE01+NA1056" AND "01_PushButton"."SE01+NA2036" AND "01_PushButton"."SE01+NA3025" AND "01_PushButton"."SE01+NA3026" AND "01_PushButton"."SC00+UC224.VS019" AND "01_PushButton"."SE01+NA2033" AND "01_PushButton"."SE01+NA2034" AND "01_PushButton"."SE01+NA2035" AND "01_PushButton"."SE01+NA1047" AND "01_PushButton"."SE01+NA1048" AND "01_PushButton"."SE01+NA1049" AND "01_PushButton"."SE01+NA1050" AND "01_PushButton"."SE01+NA1051" AND "01_PushButton"."SE01+NA2032" AND "01_PushButton"."SC00+UC214.VS019" AND "01_PushButton"."SE01+NA2029" AND "01_PushButton"."SE01+NA2030" AND "01_PushButton"."SE01+NA2031" AND "01_PushButton"."SE01+NA1041" AND "01_PushButton"."SE01+NA1042" AND "01_PushButton"."SE01+NA1043" AND "01_PushButton"."SE01+NA1044" AND "01_PushButton"."SE01+NA1045" AND "01_PushButton"."SE01+NA2028" AND "01_PushButton"."SE01+NA2075" AND "01_PushButton"."SE01+NA2077" AND "01_PushButton"."SE01+NA3030" AND "01_PushButton"."SE01+NA3031" AND "01_PushButton"."SE01+NA1120" AND "01_PushButton"."SE01+NA1121" AND "01_PushButton"."SE01+NA1119" AND "01_PushButton"."SE01+NA1118" AND "01_PushButton"."SE01+NA1117" AND "01_PushButton"."SE01+NA1116" AND "01_PushButton"."SE01+NA1115" AND "01_PushButton"."SE01+NA1114" AND "01_PushButton"."SE01+NA1113" AND "01_PushButton"."SE01+NA1112" AND "01_PushButton"."SE01+NA1125" AND "01_PushButton"."SE01+NA1126" AND "01_PushButton"."SE01+NA1103" AND "01_PushButton"."SE01+NA1104" AND "01_PushButton"."SE01+FIRE" AND "01_PushButton"."SE01+NA1131" AND "01_PushButton"."SE01+NA1129" AND "01_PushButton"."SE01+NA1130" AND "01_PushButton"."SE01+NA1132" AND "01_PushButton".FALSE AND "01_PushButton".FALSE AND "01_PushButton".FALSE AND "01_PushButton".FALSE AND "01_PushButton".FALSE AND "01_PushButton".FALSE AND "01_PushButton".FALSE AND "01_PushButton".FALSE AND "01_PushButton".FALSE AND "01_PushButton".FALSE AND "01_PushButton".FALSE AND "01_PushButton".FALSE AND "01_PushButton".FALSE AND "01_PushButton".FALSE AND "01_PushButton".FALSE AND "01_PushButton".FALSE AND "01_PushButton".FALSE AND "01_PushButton".FALSE AND "01_PushButton".FALSE AND "01_PushButton".FALSE AND "01_PushButton".FALSE AND "01_PushButton".FALSE AND "01_PushButton".FALSE AND "01_PushButton".FALSE AND "01_PushButton".FALSE AND "01_PushButton".FALSE AND "01_PushButton".FALSE AND "01_PushButton".FALSE AND "01_PushButton".FALSE AND "01_PushButton".FALSE AND "01_PushButton".FALSE AND "01_PushButton".FALSE AND "01_PushButton".FALSE AND "01_PushButton".FALSE AND "01_PushButton".FALSE AND "01_PushButton".FALSE AND "01_PushButton".FALSE AND "01_PushButton".FALSE AND "01_PushButton".FALSE AND "01_PushButton".FALSE AND "01_PushButton".FALSE AND "01_PushButton".FALSE AND "01_PushButton".FALSE AND "01_PushButton".FALSE AND "01_PushButton".FALSE AND "01_PushButton".FALSE AND "01_PushButton".FALSE AND "01_PushButton".FALSE AND "01_PushButton".FALSE AND "01_PushButton".FALSE AND "01_PushButton".FALSE AND "01_PushButton".FALSE AND "01_PushButton".FALSE AND "01_PushButton".FALSE AND "01_PushButton".FALSE AND "01_PushButton".FALSE AND "01_PushButton".FALSE AND "01_PushButton".FALSE AND "01_PushButton".FALSE AND "01_PushButton".FALSE AND "01_PushButton".FALSE AND "01_PushButton".FALSE AND "01_PushButton".FALSE AND "01_PushButton".FALSE AND "01_PushButton".FALSE AND "01_PushButton".FALSE AND "01_PushButton".FALSE AND "01_PushButton".FALSE AND "01_PushButton".FALSE AND "01_PushButton".FALSE AND "01_PushButton".FALSE AND "01_PushButton".FALSE AND "01_PushButton".FALSE AND "01_PushButton".FALSE AND "01_PushButton".FALSE AND "01_PushButton".FALSE AND "01_PushButton".FALSE AND "01_PushButton".FALSE AND "01_PushButton".FALSE AND "01_PushButton".FALSE AND "01_PushButton".FALSE AND "01_PushButton".FALSE AND "01_PushButton".FALSE AND "01_PushButton".FALSE AND "01_PushButton".FALSE AND "01_PushButton".FALSE AND "01_PushButton".FALSE AND "01_PushButton".FALSE AND "01_PushButton".FALSE AND "01_PushButton".FALSE AND "01_PushButton".FALSE AND "01_PushButton".FALSE AND "01_PushButton".FALSE AND "01_PushButton".FALSE AND "01_PushButton".FALSE AND "01_PushButton".FALSE AND "01_PushButton".FALSE AND "01_PushButton".FALSE AND "01_PushButton".FALSE AND "01_PushButton".FALSE AND "01_PushButton".FALSE AND "01_PushButton".FALSE AND "01_PushButton".FALSE AND "01_PushButton".FALSE AND "01_PushButton".FALSE AND "01_PushButton".FALSE AND "01_PushButton".FALSE AND "01_PushButton".FALSE AND "01_PushButton".FALSE AND "01_PushButton".FALSE AND "01_PushButton".FALSE AND "01_PushButton".FALSE AND "01_PushButton".FALSE AND "01_PushButton".FALSE AND "01_PushButton".FALSE AND "01_PushButton".FALSE AND "01_PushButton".FALSE AND "01_PushButton".FALSE AND "01_PushButton".FALSE AND "01_PushButton".FALSE AND "01_PushButton".FALSE AND "01_PushButton".FALSE AND "01_PushButton".FALSE AND "01_PushButton".FALSE AND "01_PushButton".FALSE AND "01_PushButton".FALSE AND "01_PushButton".FALSE AND "01_PushButton".FALSE AND "01_PushButton".FALSE AND "01_PushButton".FALSE AND "01_PushButton".FALSE AND "01_PushButton".FALSE AND "01_PushButton".FALSE AND "01_PushButton".FALSE AND "01_PushButton".FALSE AND "01_PushButton".FALSE AND "01_PushButton".FALSE AND "01_PushButton".FALSE AND "01_PushButton".FALSE AND "01_PushButton".FALSE AND "01_PushButton".FALSE AND "01_PushButton".FALSE AND "01_PushButton".FALSE AND "01_PushButton".FALSE AND "01_PushButton".FALSE AND "01_PushButton".FALSE AND "01_PushButton".FALSE AND "01_PushButton".FALSE AND "01_PushButton".FALSE AND "01_PushButton".FALSE AND "01_PushButton".FALSE AND "01_PushButton".FALSE AND "01_PushButton".FALSE AND "01_PushButton".FALSE AND "01_PushButton".FALSE AND "01_PushButton".FALSE AND "01_PushButton".FALSE AND "01_PushButton".FALSE AND "01_PushButton".FALSE AND "01_PushButton".FALSE AND "01_PushButton".FALSE AND "01_PushButton".FALSE AND "01_PushButton".FALSE AND "01_PushButton".FALSE AND "01_PushButton".FALSE AND "01_PushButton".FALSE AND "01_PushButton".FALSE AND "01_PushButton".FALSE AND "01_PushButton".FALSE AND "01_PushButton".FALSE AND "01_PushButton".FALSE AND "01_PushButton".FALSE AND "01_PushButton".FALSE AND "01_PushButton".FALSE AND "01_PushButton".FALSE AND "01_PushButton".FALSE AND "01_PushButton".FALSE AND "01_PushButton".FALSE AND "01_PushButton".FALSE AND "01_PushButton".FALSE AND "01_PushButton".FALSE AND "01_PushButton".FALSE AND "01_PushButton".FALSE AND "01_PushButton".FALSE AND "01_PushButton".FALSE AND "01_PushButton".FALSE AND "01_PushButton".FALSE AND "01_PushButton".FALSE AND "01_PushButton".FALSE AND "01_PushButton".FALSE AND "01_PushButton".FALSE AND "01_PushButton".FALSE AND "01_PushButton".FALSE AND "01_PushButton".FALSE AND "01_PushButton".FALSE AND "01_PushButton".FALSE AND "01_PushButton".FALSE AND "01_PushButton".FALSE AND "01_PushButton".FALSE AND "01_PushButton".FALSE AND "01_PushButton".FALSE AND "01_PushButton".FALSE AND "01_PushButton".FALSE AND "01_PushButton".FALSE AND "01_PushButton".FALSE AND "01_PushButton".FALSE AND "01_PushButton".FALSE AND "01_PushButton".FALSE AND "01_PushButton".FALSE AND "01_PushButton".FALSE AND "01_PushButton".FALSE AND "01_PushButton".FALSE AND "01_PushButton".FALSE AND "01_PushButton".FALSE AND "01_PushButton".FALSE AND "01_PushButton".FALSE AND "01_PushButton".FALSE AND "01_PushButton".FALSE AND "01_PushButton".FALSE AND "01_PushButton".FALSE AND "01_PushButton".FALSE AND "01_PushButton".FALSE AND "01_PushButton".FALSE AND "01_PushButton".FALSE AND "01_PushButton".FALSE AND "01_PushButton".FALSE AND "01_PushButton".FALSE AND "01_PushButton".FALSE AND "01_PushButton".FALSE AND "01_PushButton".FALSE AND "01_PushButton".FALSE AND "01_PushButton".FALSE AND "01_PushButton".FALSE AND "01_PushButton".FALSE AND "01_PushButton".FALSE AND "01_PushButton".FALSE AND "01_PushButton".FALSE AND "01_PushButton".FALSE AND "01_PushButton".FALSE AND "01_PushButton".FALSE AND "01_PushButton".FALSE AND "01_PushButton".FALSE AND "01_PushButton".FALSE AND "01_PushButton".FALSE;
END_REGION

REGION Network 3: S3 PB - ^S3 | Sorter FLY Upper [=SF03]
   // 51 - 250 Inputs
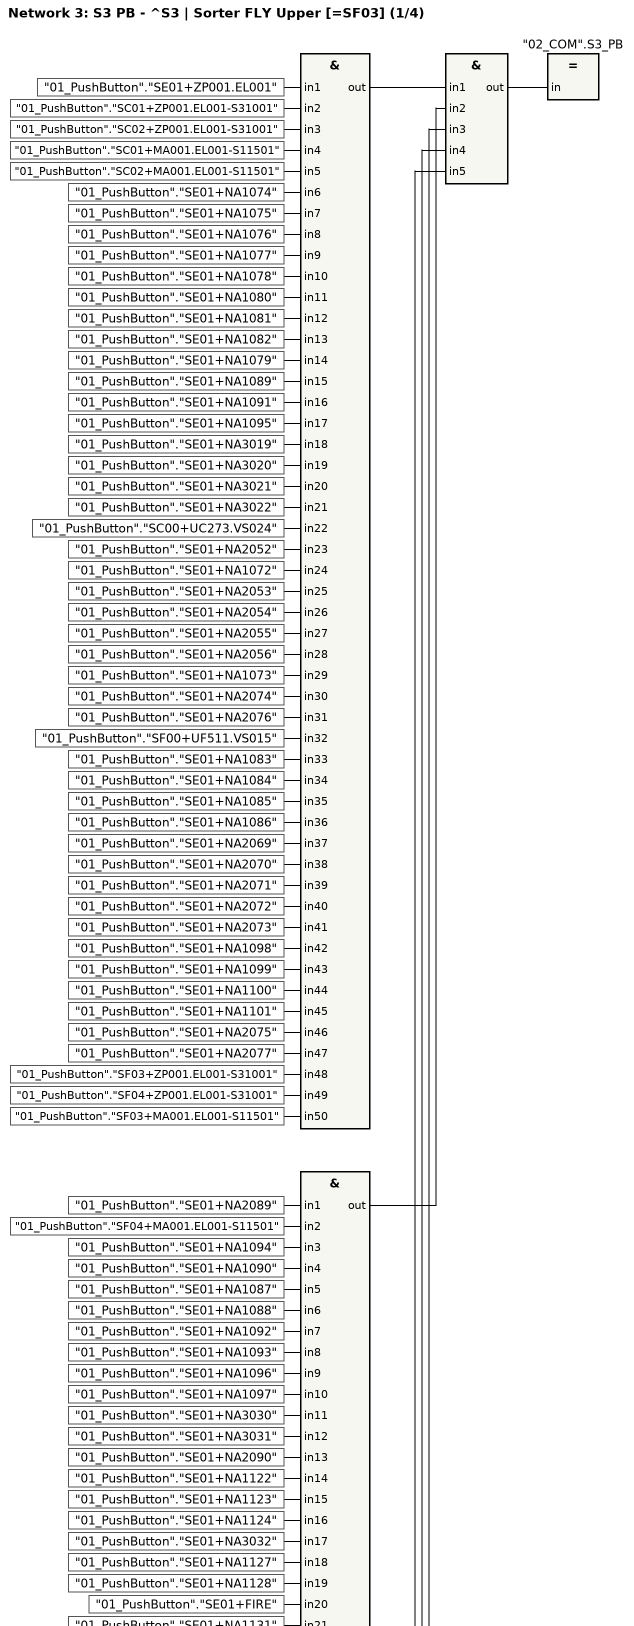
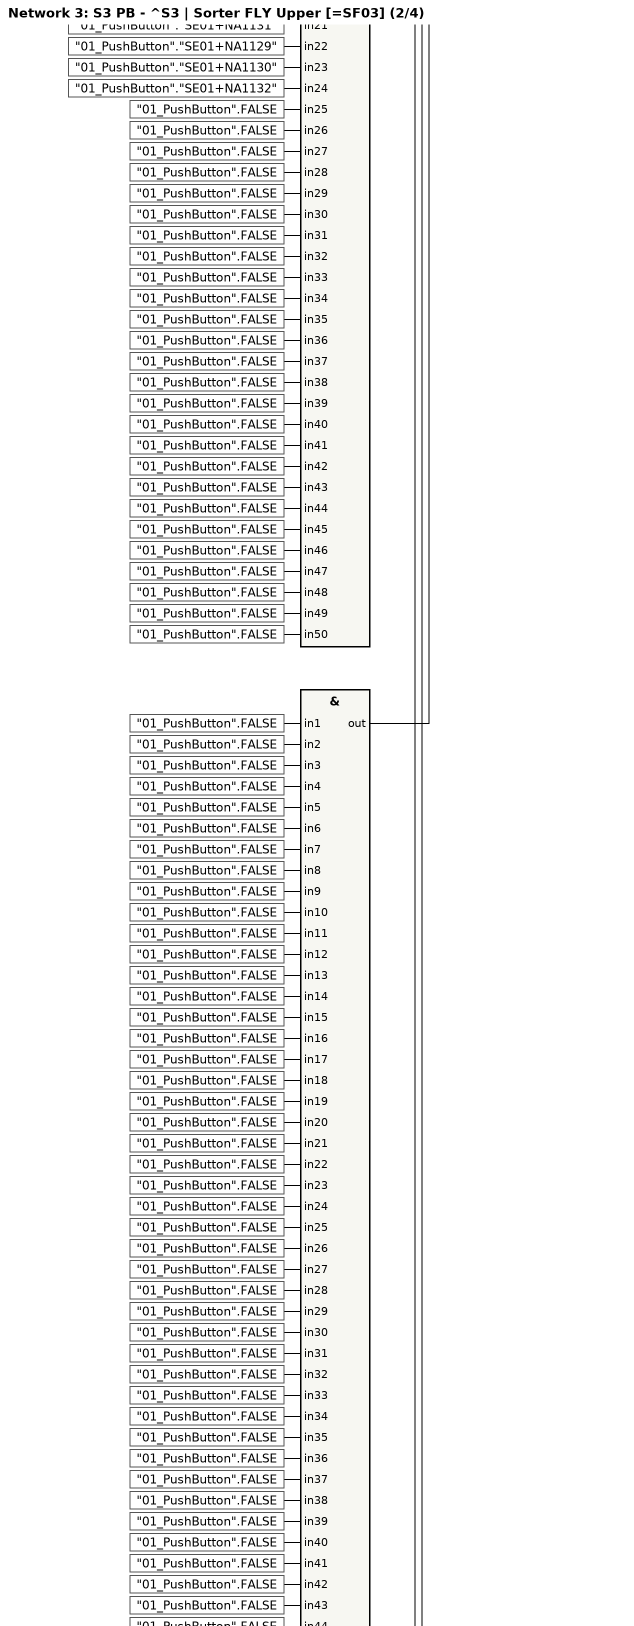
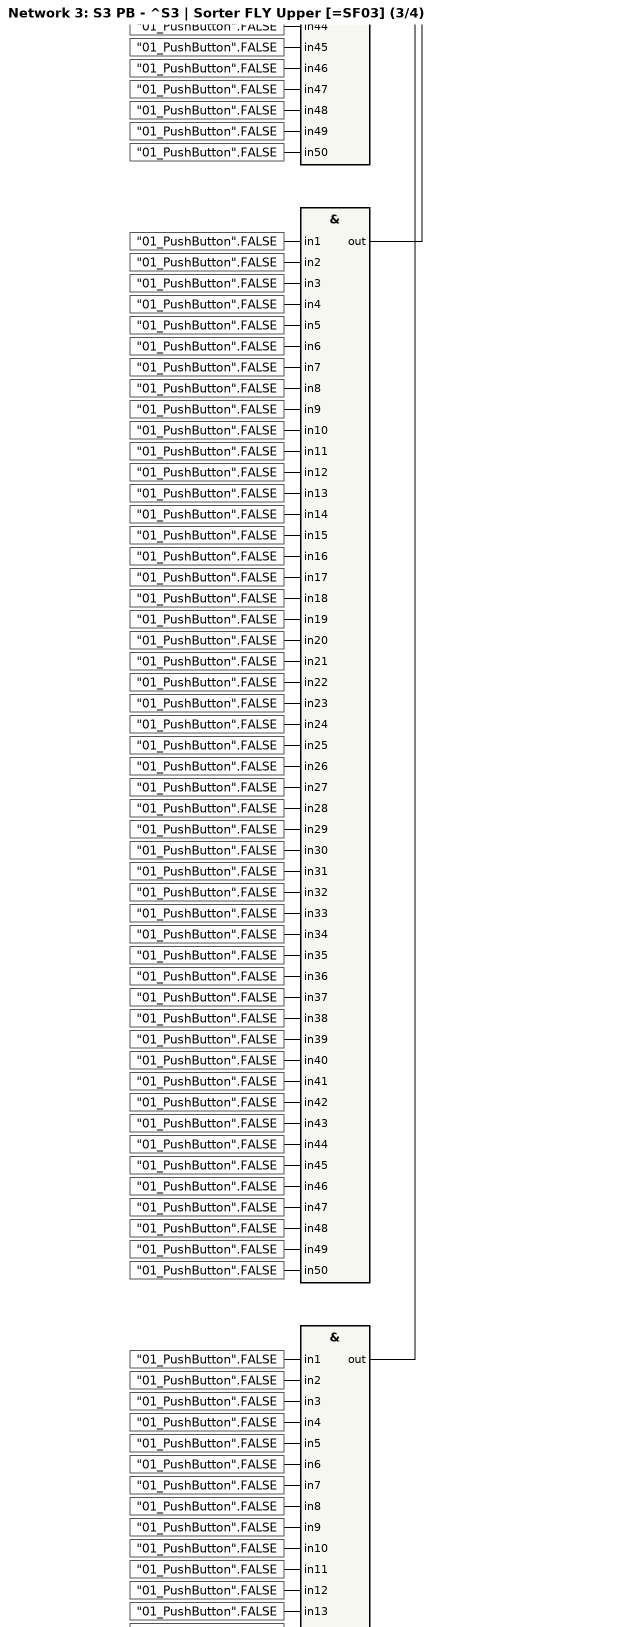
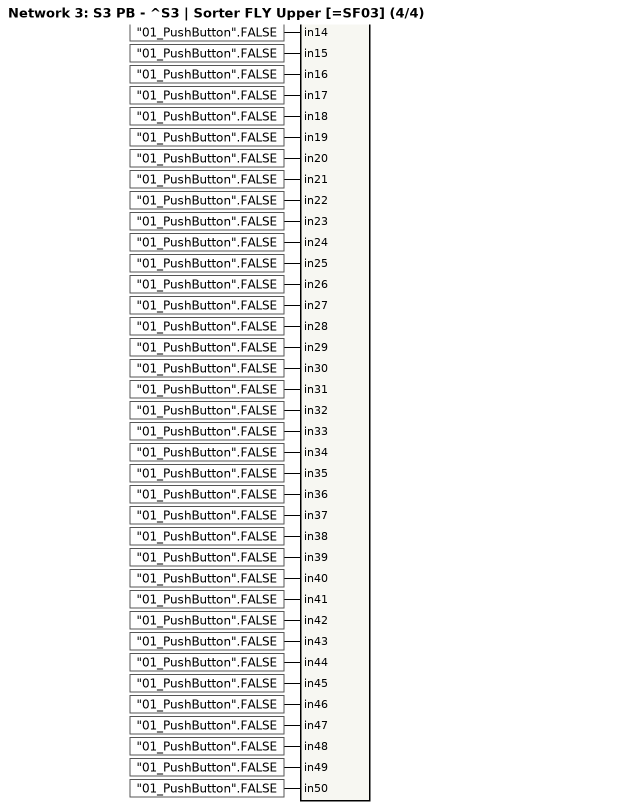
   "02_COM".S3_PB := "01_PushButton"."SE01+ZP001.EL001" AND "01_PushButton"."SC01+ZP001.EL001-S31001" AND "01_PushButton"."SC02+ZP001.EL001-S31001" AND "01_PushButton"."SC01+MA001.EL001-S11501" AND "01_PushButton"."SC02+MA001.EL001-S11501" AND "01_PushButton"."SE01+NA1074" AND "01_PushButton"."SE01+NA1075" AND "01_PushButton"."SE01+NA1076" AND "01_PushButton"."SE01+NA1077" AND "01_PushButton"."SE01+NA1078" AND "01_PushButton"."SE01+NA1080" AND "01_PushButton"."SE01+NA1081" AND "01_PushButton"."SE01+NA1082" AND "01_PushButton"."SE01+NA1079" AND "01_PushButton"."SE01+NA1089" AND "01_PushButton"."SE01+NA1091" AND "01_PushButton"."SE01+NA1095" AND "01_PushButton"."SE01+NA3019" AND "01_PushButton"."SE01+NA3020" AND "01_PushButton"."SE01+NA3021" AND "01_PushButton"."SE01+NA3022" AND "01_PushButton"."SC00+UC273.VS024" AND "01_PushButton"."SE01+NA2052" AND "01_PushButton"."SE01+NA1072" AND "01_PushButton"."SE01+NA2053" AND "01_PushButton"."SE01+NA2054" AND "01_PushButton"."SE01+NA2055" AND "01_PushButton"."SE01+NA2056" AND "01_PushButton"."SE01+NA1073" AND "01_PushButton"."SE01+NA2074" AND "01_PushButton"."SE01+NA2076" AND "01_PushButton"."SF00+UF511.VS015" AND "01_PushButton"."SE01+NA1083" AND "01_PushButton"."SE01+NA1084" AND "01_PushButton"."SE01+NA1085" AND "01_PushButton"."SE01+NA1086" AND "01_PushButton"."SE01+NA2069" AND "01_PushButton"."SE01+NA2070" AND "01_PushButton"."SE01+NA2071" AND "01_PushButton"."SE01+NA2072" AND "01_PushButton"."SE01+NA2073" AND "01_PushButton"."SE01+NA1098" AND "01_PushButton"."SE01+NA1099" AND "01_PushButton"."SE01+NA1100" AND "01_PushButton"."SE01+NA1101" AND "01_PushButton"."SE01+NA2075" AND "01_PushButton"."SE01+NA2077" AND "01_PushButton"."SF03+ZP001.EL001-S31001" AND "01_PushButton"."SF04+ZP001.EL001-S31001" AND "01_PushButton"."SF03+MA001.EL001-S11501" AND "01_PushButton"."SE01+NA2089" AND "01_PushButton"."SF04+MA001.EL001-S11501" AND "01_PushButton"."SE01+NA1094" AND "01_PushButton"."SE01+NA1090" AND "01_PushButton"."SE01+NA1087" AND "01_PushButton"."SE01+NA1088" AND "01_PushButton"."SE01+NA1092" AND "01_PushButton"."SE01+NA1093" AND "01_PushButton"."SE01+NA1096" AND "01_PushButton"."SE01+NA1097" AND "01_PushButton"."SE01+NA3030" AND "01_PushButton"."SE01+NA3031" AND "01_PushButton"."SE01+NA2090" AND "01_PushButton"."SE01+NA1122" AND "01_PushButton"."SE01+NA1123" AND "01_PushButton"."SE01+NA1124" AND "01_PushButton"."SE01+NA3032" AND "01_PushButton"."SE01+NA1127" AND "01_PushButton"."SE01+NA1128" AND "01_PushButton"."SE01+FIRE" AND "01_PushButton"."SE01+NA1131" AND "01_PushButton"."SE01+NA1129" AND "01_PushButton"."SE01+NA1130" AND "01_PushButton"."SE01+NA1132" AND "01_PushButton".FALSE AND "01_PushButton".FALSE AND "01_PushButton".FALSE AND "01_PushButton".FALSE AND "01_PushButton".FALSE AND "01_PushButton".FALSE AND "01_PushButton".FALSE AND "01_PushButton".FALSE AND "01_PushButton".FALSE AND "01_PushButton".FALSE AND "01_PushButton".FALSE AND "01_PushButton".FALSE AND "01_PushButton".FALSE AND "01_PushButton".FALSE AND "01_PushButton".FALSE AND "01_PushButton".FALSE AND "01_PushButton".FALSE AND "01_PushButton".FALSE AND "01_PushButton".FALSE AND "01_PushButton".FALSE AND "01_PushButton".FALSE AND "01_PushButton".FALSE AND "01_PushButton".FALSE AND "01_PushButton".FALSE AND "01_PushButton".FALSE AND "01_PushButton".FALSE AND "01_PushButton".FALSE AND "01_PushButton".FALSE AND "01_PushButton".FALSE AND "01_PushButton".FALSE AND "01_PushButton".FALSE AND "01_PushButton".FALSE AND "01_PushButton".FALSE AND "01_PushButton".FALSE AND "01_PushButton".FALSE AND "01_PushButton".FALSE AND "01_PushButton".FALSE AND "01_PushButton".FALSE AND "01_PushButton".FALSE AND "01_PushButton".FALSE AND "01_PushButton".FALSE AND "01_PushButton".FALSE AND "01_PushButton".FALSE AND "01_PushButton".FALSE AND "01_PushButton".FALSE AND "01_PushButton".FALSE AND "01_PushButton".FALSE AND "01_PushButton".FALSE AND "01_PushButton".FALSE AND "01_PushButton".FALSE AND "01_PushButton".FALSE AND "01_PushButton".FALSE AND "01_PushButton".FALSE AND "01_PushButton".FALSE AND "01_PushButton".FALSE AND "01_PushButton".FALSE AND "01_PushButton".FALSE AND "01_PushButton".FALSE AND "01_PushButton".FALSE AND "01_PushButton".FALSE AND "01_PushButton".FALSE AND "01_PushButton".FALSE AND "01_PushButton".FALSE AND "01_PushButton".FALSE AND "01_PushButton".FALSE AND "01_PushButton".FALSE AND "01_PushButton".FALSE AND "01_PushButton".FALSE AND "01_PushButton".FALSE AND "01_PushButton".FALSE AND "01_PushButton".FALSE AND "01_PushButton".FALSE AND "01_PushButton".FALSE AND "01_PushButton".FALSE AND "01_PushButton".FALSE AND "01_PushButton".FALSE AND "01_PushButton".FALSE AND "01_PushButton".FALSE AND "01_PushButton".FALSE AND "01_PushButton".FALSE AND "01_PushButton".FALSE AND "01_PushButton".FALSE AND "01_PushButton".FALSE AND "01_PushButton".FALSE AND "01_PushButton".FALSE AND "01_PushButton".FALSE AND "01_PushButton".FALSE AND "01_PushButton".FALSE AND "01_PushButton".FALSE AND "01_PushButton".FALSE AND "01_PushButton".FALSE AND "01_PushButton".FALSE AND "01_PushButton".FALSE AND "01_PushButton".FALSE AND "01_PushButton".FALSE AND "01_PushButton".FALSE AND "01_PushButton".FALSE AND "01_PushButton".FALSE AND "01_PushButton".FALSE AND "01_PushButton".FALSE AND "01_PushButton".FALSE AND "01_PushButton".FALSE AND "01_PushButton".FALSE AND "01_PushButton".FALSE AND "01_PushButton".FALSE AND "01_PushButton".FALSE AND "01_PushButton".FALSE AND "01_PushButton".FALSE AND "01_PushButton".FALSE AND "01_PushButton".FALSE AND "01_PushButton".FALSE AND "01_PushButton".FALSE AND "01_PushButton".FALSE AND "01_PushButton".FALSE AND "01_PushButton".FALSE AND "01_PushButton".FALSE AND "01_PushButton".FALSE AND "01_PushButton".FALSE AND "01_PushButton".FALSE AND "01_PushButton".FALSE AND "01_PushButton".FALSE AND "01_PushButton".FALSE AND "01_PushButton".FALSE AND "01_PushButton".FALSE AND "01_PushButton".FALSE AND "01_PushButton".FALSE AND "01_PushButton".FALSE AND "01_PushButton".FALSE AND "01_PushButton".FALSE AND "01_PushButton".FALSE AND "01_PushButton".FALSE AND "01_PushButton".FALSE AND "01_PushButton".FALSE AND "01_PushButton".FALSE AND "01_PushButton".FALSE AND "01_PushButton".FALSE AND "01_PushButton".FALSE AND "01_PushButton".FALSE AND "01_PushButton".FALSE AND "01_PushButton".FALSE AND "01_PushButton".FALSE AND "01_PushButton".FALSE AND "01_PushButton".FALSE AND "01_PushButton".FALSE AND "01_PushButton".FALSE AND "01_PushButton".FALSE AND "01_PushButton".FALSE AND "01_PushButton".FALSE AND "01_PushButton".FALSE AND "01_PushButton".FALSE AND "01_PushButton".FALSE AND "01_PushButton".FALSE AND "01_PushButton".FALSE AND "01_PushButton".FALSE AND "01_PushButton".FALSE AND "01_PushButton".FALSE AND "01_PushButton".FALSE AND "01_PushButton".FALSE AND "01_PushButton".FALSE AND "01_PushButton".FALSE AND "01_PushButton".FALSE AND "01_PushButton".FALSE AND "01_PushButton".FALSE AND "01_PushButton".FALSE AND "01_PushButton".FALSE AND "01_PushButton".FALSE AND "01_PushButton".FALSE AND "01_PushButton".FALSE AND "01_PushButton".FALSE AND "01_PushButton".FALSE AND "01_PushButton".FALSE AND "01_PushButton".FALSE AND "01_PushButton".FALSE AND "01_PushButton".FALSE AND "01_PushButton".FALSE AND "01_PushButton".FALSE;
END_REGION

REGION Network 4: S4 PB - ^S4 | Sorter COY Upper [=SC01]
   // 51 - 250 Inputs
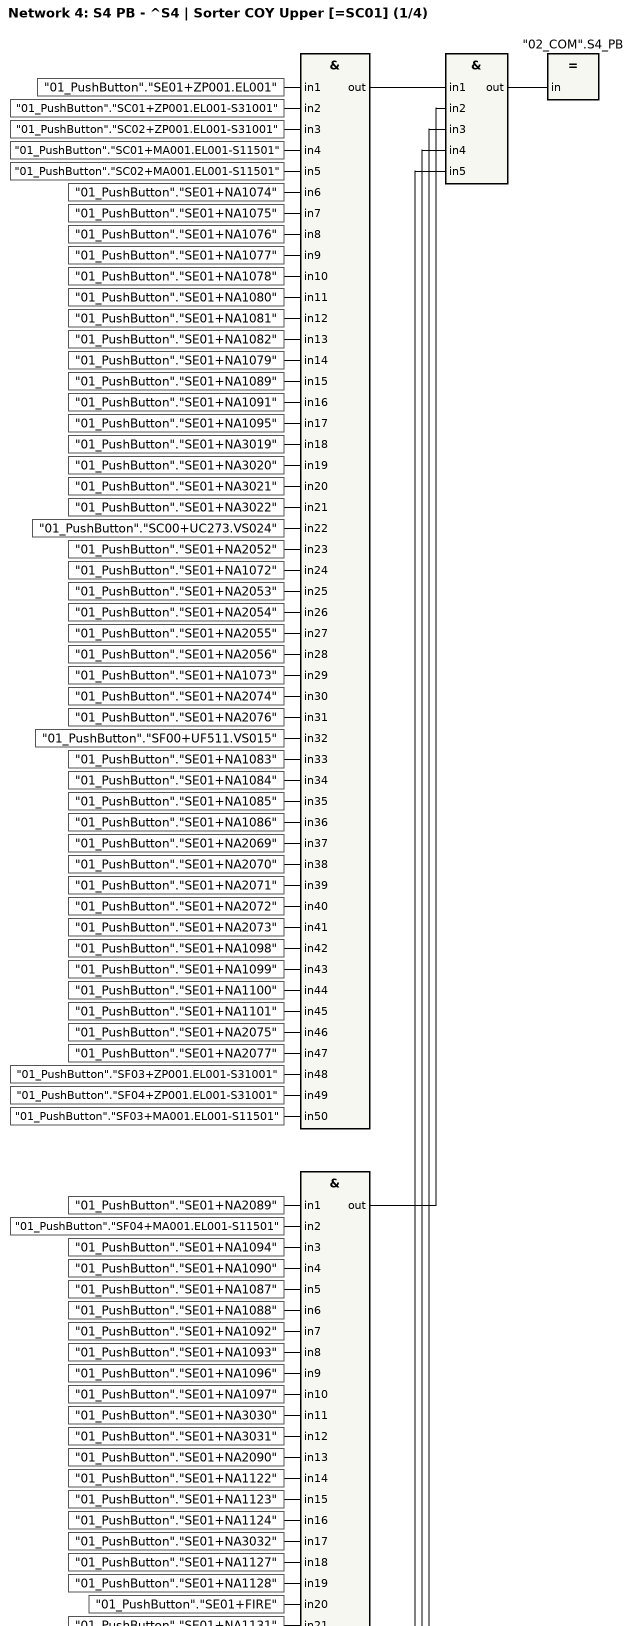
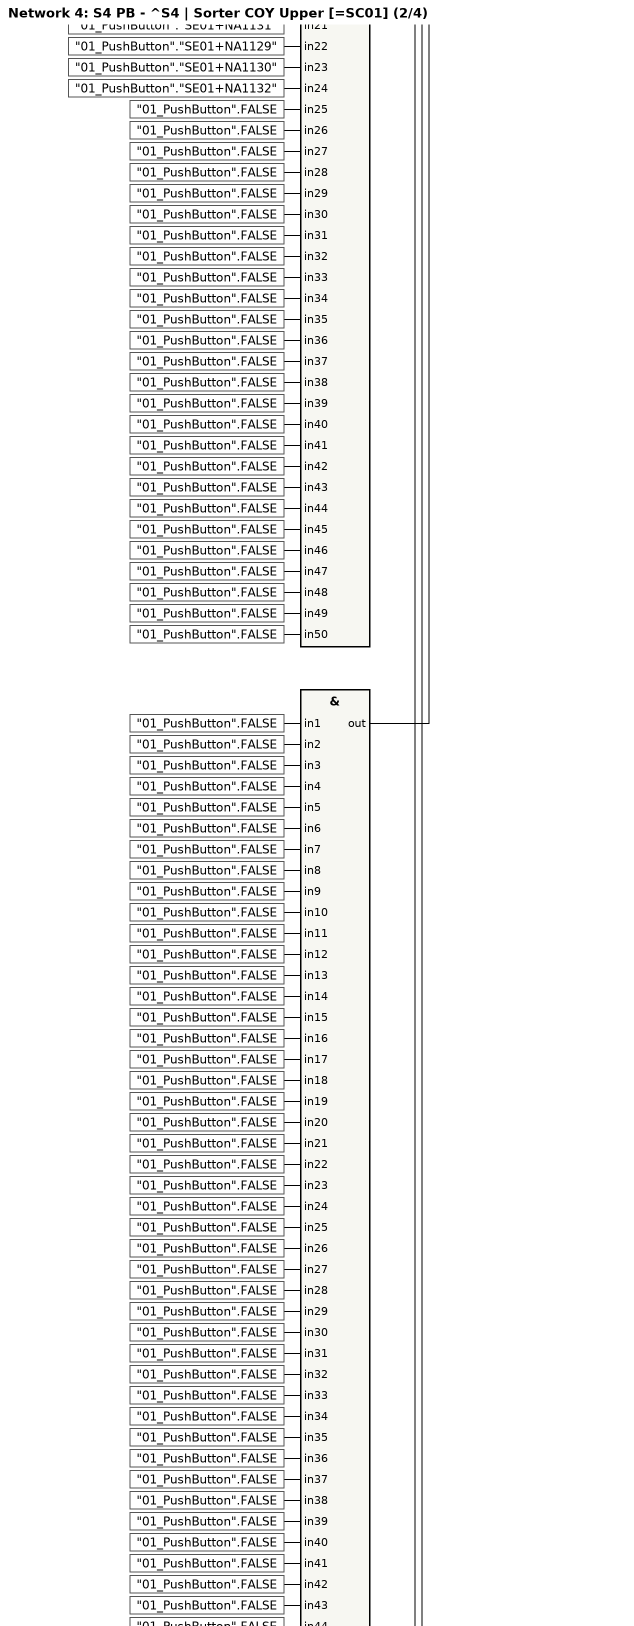
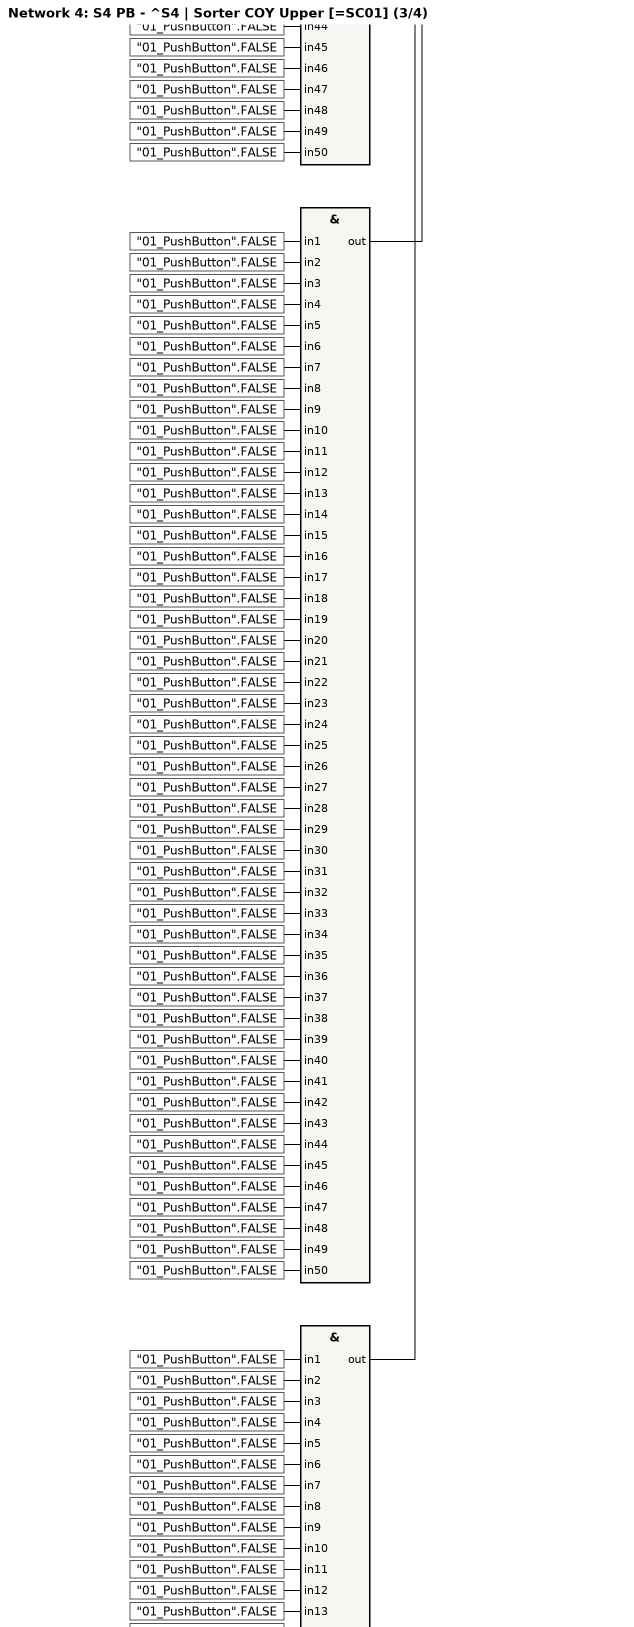
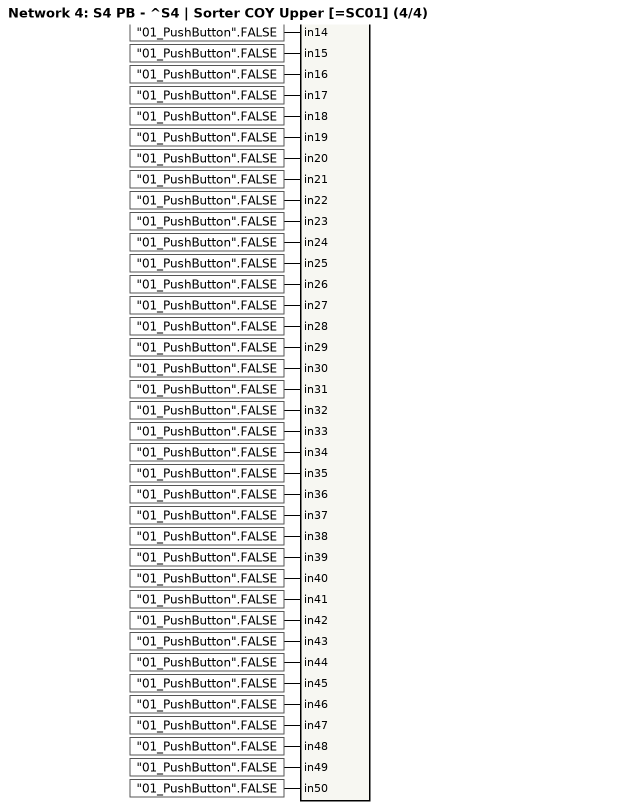
   "02_COM".S4_PB := "01_PushButton"."SE01+ZP001.EL001" AND "01_PushButton"."SC01+ZP001.EL001-S31001" AND "01_PushButton"."SC02+ZP001.EL001-S31001" AND "01_PushButton"."SC01+MA001.EL001-S11501" AND "01_PushButton"."SC02+MA001.EL001-S11501" AND "01_PushButton"."SE01+NA1074" AND "01_PushButton"."SE01+NA1075" AND "01_PushButton"."SE01+NA1076" AND "01_PushButton"."SE01+NA1077" AND "01_PushButton"."SE01+NA1078" AND "01_PushButton"."SE01+NA1080" AND "01_PushButton"."SE01+NA1081" AND "01_PushButton"."SE01+NA1082" AND "01_PushButton"."SE01+NA1079" AND "01_PushButton"."SE01+NA1089" AND "01_PushButton"."SE01+NA1091" AND "01_PushButton"."SE01+NA1095" AND "01_PushButton"."SE01+NA3019" AND "01_PushButton"."SE01+NA3020" AND "01_PushButton"."SE01+NA3021" AND "01_PushButton"."SE01+NA3022" AND "01_PushButton"."SC00+UC273.VS024" AND "01_PushButton"."SE01+NA2052" AND "01_PushButton"."SE01+NA1072" AND "01_PushButton"."SE01+NA2053" AND "01_PushButton"."SE01+NA2054" AND "01_PushButton"."SE01+NA2055" AND "01_PushButton"."SE01+NA2056" AND "01_PushButton"."SE01+NA1073" AND "01_PushButton"."SE01+NA2074" AND "01_PushButton"."SE01+NA2076" AND "01_PushButton"."SF00+UF511.VS015" AND "01_PushButton"."SE01+NA1083" AND "01_PushButton"."SE01+NA1084" AND "01_PushButton"."SE01+NA1085" AND "01_PushButton"."SE01+NA1086" AND "01_PushButton"."SE01+NA2069" AND "01_PushButton"."SE01+NA2070" AND "01_PushButton"."SE01+NA2071" AND "01_PushButton"."SE01+NA2072" AND "01_PushButton"."SE01+NA2073" AND "01_PushButton"."SE01+NA1098" AND "01_PushButton"."SE01+NA1099" AND "01_PushButton"."SE01+NA1100" AND "01_PushButton"."SE01+NA1101" AND "01_PushButton"."SE01+NA2075" AND "01_PushButton"."SE01+NA2077" AND "01_PushButton"."SF03+ZP001.EL001-S31001" AND "01_PushButton"."SF04+ZP001.EL001-S31001" AND "01_PushButton"."SF03+MA001.EL001-S11501" AND "01_PushButton"."SE01+NA2089" AND "01_PushButton"."SF04+MA001.EL001-S11501" AND "01_PushButton"."SE01+NA1094" AND "01_PushButton"."SE01+NA1090" AND "01_PushButton"."SE01+NA1087" AND "01_PushButton"."SE01+NA1088" AND "01_PushButton"."SE01+NA1092" AND "01_PushButton"."SE01+NA1093" AND "01_PushButton"."SE01+NA1096" AND "01_PushButton"."SE01+NA1097" AND "01_PushButton"."SE01+NA3030" AND "01_PushButton"."SE01+NA3031" AND "01_PushButton"."SE01+NA2090" AND "01_PushButton"."SE01+NA1122" AND "01_PushButton"."SE01+NA1123" AND "01_PushButton"."SE01+NA1124" AND "01_PushButton"."SE01+NA3032" AND "01_PushButton"."SE01+NA1127" AND "01_PushButton"."SE01+NA1128" AND "01_PushButton"."SE01+FIRE" AND "01_PushButton"."SE01+NA1131" AND "01_PushButton"."SE01+NA1129" AND "01_PushButton"."SE01+NA1130" AND "01_PushButton"."SE01+NA1132" AND "01_PushButton".FALSE AND "01_PushButton".FALSE AND "01_PushButton".FALSE AND "01_PushButton".FALSE AND "01_PushButton".FALSE AND "01_PushButton".FALSE AND "01_PushButton".FALSE AND "01_PushButton".FALSE AND "01_PushButton".FALSE AND "01_PushButton".FALSE AND "01_PushButton".FALSE AND "01_PushButton".FALSE AND "01_PushButton".FALSE AND "01_PushButton".FALSE AND "01_PushButton".FALSE AND "01_PushButton".FALSE AND "01_PushButton".FALSE AND "01_PushButton".FALSE AND "01_PushButton".FALSE AND "01_PushButton".FALSE AND "01_PushButton".FALSE AND "01_PushButton".FALSE AND "01_PushButton".FALSE AND "01_PushButton".FALSE AND "01_PushButton".FALSE AND "01_PushButton".FALSE AND "01_PushButton".FALSE AND "01_PushButton".FALSE AND "01_PushButton".FALSE AND "01_PushButton".FALSE AND "01_PushButton".FALSE AND "01_PushButton".FALSE AND "01_PushButton".FALSE AND "01_PushButton".FALSE AND "01_PushButton".FALSE AND "01_PushButton".FALSE AND "01_PushButton".FALSE AND "01_PushButton".FALSE AND "01_PushButton".FALSE AND "01_PushButton".FALSE AND "01_PushButton".FALSE AND "01_PushButton".FALSE AND "01_PushButton".FALSE AND "01_PushButton".FALSE AND "01_PushButton".FALSE AND "01_PushButton".FALSE AND "01_PushButton".FALSE AND "01_PushButton".FALSE AND "01_PushButton".FALSE AND "01_PushButton".FALSE AND "01_PushButton".FALSE AND "01_PushButton".FALSE AND "01_PushButton".FALSE AND "01_PushButton".FALSE AND "01_PushButton".FALSE AND "01_PushButton".FALSE AND "01_PushButton".FALSE AND "01_PushButton".FALSE AND "01_PushButton".FALSE AND "01_PushButton".FALSE AND "01_PushButton".FALSE AND "01_PushButton".FALSE AND "01_PushButton".FALSE AND "01_PushButton".FALSE AND "01_PushButton".FALSE AND "01_PushButton".FALSE AND "01_PushButton".FALSE AND "01_PushButton".FALSE AND "01_PushButton".FALSE AND "01_PushButton".FALSE AND "01_PushButton".FALSE AND "01_PushButton".FALSE AND "01_PushButton".FALSE AND "01_PushButton".FALSE AND "01_PushButton".FALSE AND "01_PushButton".FALSE AND "01_PushButton".FALSE AND "01_PushButton".FALSE AND "01_PushButton".FALSE AND "01_PushButton".FALSE AND "01_PushButton".FALSE AND "01_PushButton".FALSE AND "01_PushButton".FALSE AND "01_PushButton".FALSE AND "01_PushButton".FALSE AND "01_PushButton".FALSE AND "01_PushButton".FALSE AND "01_PushButton".FALSE AND "01_PushButton".FALSE AND "01_PushButton".FALSE AND "01_PushButton".FALSE AND "01_PushButton".FALSE AND "01_PushButton".FALSE AND "01_PushButton".FALSE AND "01_PushButton".FALSE AND "01_PushButton".FALSE AND "01_PushButton".FALSE AND "01_PushButton".FALSE AND "01_PushButton".FALSE AND "01_PushButton".FALSE AND "01_PushButton".FALSE AND "01_PushButton".FALSE AND "01_PushButton".FALSE AND "01_PushButton".FALSE AND "01_PushButton".FALSE AND "01_PushButton".FALSE AND "01_PushButton".FALSE AND "01_PushButton".FALSE AND "01_PushButton".FALSE AND "01_PushButton".FALSE AND "01_PushButton".FALSE AND "01_PushButton".FALSE AND "01_PushButton".FALSE AND "01_PushButton".FALSE AND "01_PushButton".FALSE AND "01_PushButton".FALSE AND "01_PushButton".FALSE AND "01_PushButton".FALSE AND "01_PushButton".FALSE AND "01_PushButton".FALSE AND "01_PushButton".FALSE AND "01_PushButton".FALSE AND "01_PushButton".FALSE AND "01_PushButton".FALSE AND "01_PushButton".FALSE AND "01_PushButton".FALSE AND "01_PushButton".FALSE AND "01_PushButton".FALSE AND "01_PushButton".FALSE AND "01_PushButton".FALSE AND "01_PushButton".FALSE AND "01_PushButton".FALSE AND "01_PushButton".FALSE AND "01_PushButton".FALSE AND "01_PushButton".FALSE AND "01_PushButton".FALSE AND "01_PushButton".FALSE AND "01_PushButton".FALSE AND "01_PushButton".FALSE AND "01_PushButton".FALSE AND "01_PushButton".FALSE AND "01_PushButton".FALSE AND "01_PushButton".FALSE AND "01_PushButton".FALSE AND "01_PushButton".FALSE AND "01_PushButton".FALSE AND "01_PushButton".FALSE AND "01_PushButton".FALSE AND "01_PushButton".FALSE AND "01_PushButton".FALSE AND "01_PushButton".FALSE AND "01_PushButton".FALSE AND "01_PushButton".FALSE AND "01_PushButton".FALSE AND "01_PushButton".FALSE AND "01_PushButton".FALSE AND "01_PushButton".FALSE AND "01_PushButton".FALSE AND "01_PushButton".FALSE AND "01_PushButton".FALSE AND "01_PushButton".FALSE AND "01_PushButton".FALSE AND "01_PushButton".FALSE AND "01_PushButton".FALSE AND "01_PushButton".FALSE AND "01_PushButton".FALSE AND "01_PushButton".FALSE AND "01_PushButton".FALSE AND "01_PushButton".FALSE AND "01_PushButton".FALSE AND "01_PushButton".FALSE AND "01_PushButton".FALSE AND "01_PushButton".FALSE AND "01_PushButton".FALSE AND "01_PushButton".FALSE AND "01_PushButton".FALSE;
END_REGION

REGION Network 5: A1 PB - >A1 | AREA 1 - INTRO+UPSTREAM COY WEST
   // 51 - 250 Inputs
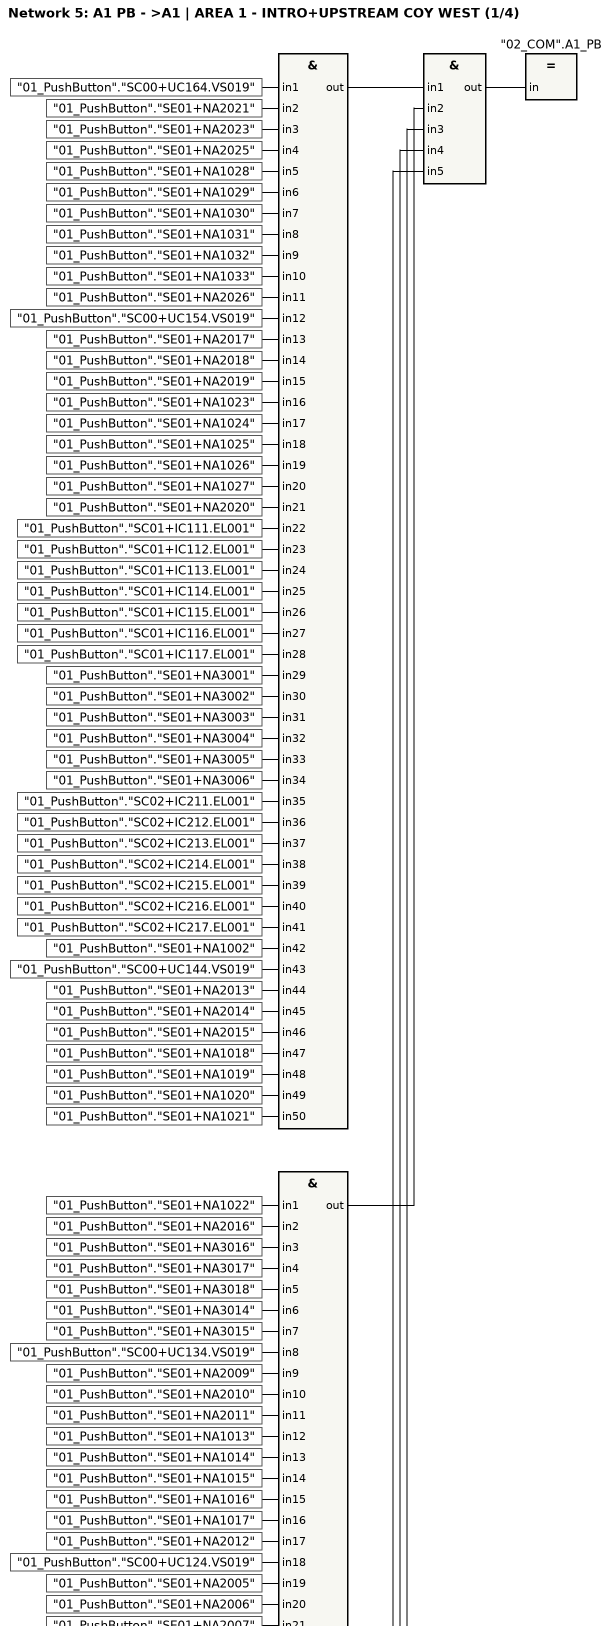
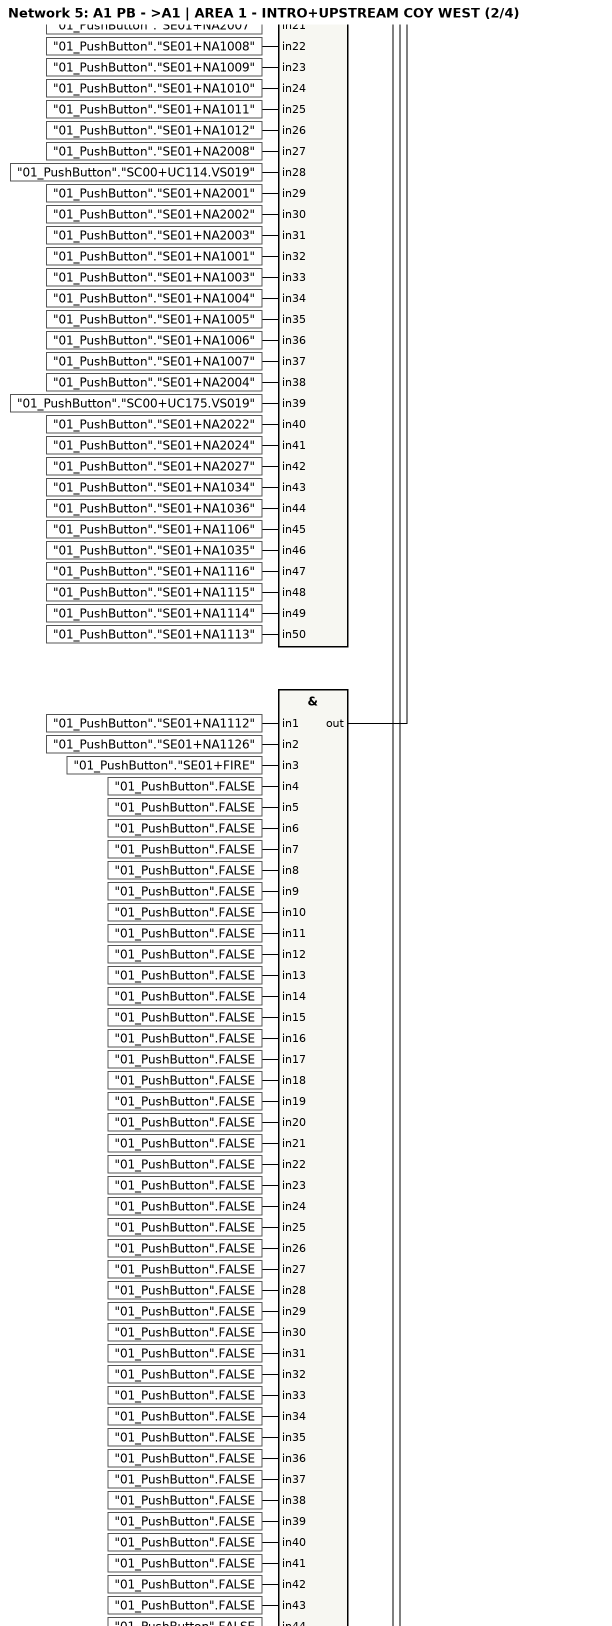
